LIN {X 0,Y 173.523,Z 389.647,A -85,B 0,C 180,E1 -26312.819,E2 -26312.819} C_VEL
LIN {X 0,Y 168.462,Z 401.528,A -85,B 0,C 180,E1 -26313.99,E2 -26313.99} C_VEL
LIN {X 0,Y 162.813,Z 412.302,A -85,B 0,C 180,E1 -26315.439,E2 -26315.439} C_VEL
LIN {X 0,Y 156.587,Z 422.141,A -85,B 0,C 180,E1 -26317.19,E2 -26317.19} C_VEL
LIN {X 0,Y 148.692,Z 432.687,A -85,B 0,C 180,E1 -26319.822,E2 -26319.822} C_VEL
LIN {X 0,Y 142.367,Z 439.895,A -85,B 0,C 180,E1 -26322.229,E2 -26322.229} C_VEL
LIN {X 0,Y 135.332,Z 447.062,A -85,B 0,C 180,E1 -26325.488,E2 -26325.488} C_VEL
LIN {X 0,Y 128.764,Z 452.875,A -85,B 0,C 180,E1 -26329.084,E2 -26329.084} C_VEL
LIN {X 0,Y 122.651,Z 457.744,A -85,B 0,C 180,E1 -26333.368,E2 -26333.368} C_VEL
LIN {X 0,Y 117.792,Z 461.088,A -85,B 0,C 180,E1 -26337.523,E2 -26337.523} C_VEL
LIN {X 0,Y 114.712,Z 462.976,A -85,B 0,C 180,E1 -26340.652,E2 -26340.652} C_VEL
LIN {X 0,Y 109.77,Z 465.505,A -85,B 0,C 180,E1 -26347.41,E2 -26347.41} C_VEL
LIN {X 0,Y 106.669,Z 466.55,A -85,B 0,C 180,E1 -26354.72,E2 -26354.72} C_VEL
LIN {X 0,Y 105.797,Z 466.508,A -85,B 0,C 180,E1 -26358.505,E2 -26358.505} C_VEL
LIN {X 0,Y 105.23,Z 465.234,A -85,B 0,C 180,E1 -26366.171,E2 -26366.171} C_VEL
LIN {X 0,Y 105.415,Z 464.016,A -85,B 0,C 180,E1 -26370,E2 -26370} C_VEL
LIN {X 0,Y 105.329,Z 461.286,A -85,B 0,C 180,E1 -26375.744,E2 -26375.744} C_VEL
LIN {X 0,Y 105.868,Z 457.47,A -85,B 0,C 180,E1 -26381.487,E2 -26381.487} C_VEL
LIN {X 0,Y 107.202,Z 452.472,A -85,B 0,C 180,E1 -26387.158,E2 -26387.158} C_VEL
LIN {X 0,Y 109.577,Z 446.168,A -85,B 0,C 180,E1 -26392.633,E2 -26392.633} C_VEL
LIN {X 0,Y 112.757,Z 438.217,A -85,B 0,C 180,E1 -26397.869,E2 -26397.869} C_VEL
LIN {X 0,Y 116.232,Z 429.754,A -85,B 0,C 180,E1 -26402.134,E2 -26402.134} C_VEL
LIN {X 0,Y 119.944,Z 420.166,A -85,B 0,C 180,E1 -26405.869,E2 -26405.869} C_VEL
LIN {X 0,Y 123.287,Z 410.655,A -85,B 0,C 180,E1 -26408.739,E2 -26408.739} C_VEL
LIN {X 0,Y 124.479,Z 405.7,A -85,B 0,C 180,E1 -26410.12,E2 -26410.12} C_VEL
LIN {X 0,Y 124.615,Z 397.297,A -85,B 0,C 180,E1 -26412.55,E2 -26412.55} C_VEL
LIN {X 0,Y 124.479,Z 388.532,A -85,B 0,C 180,E1 -26414.726,E2 -26414.726} C_VEL
LIN {X 0,Y 125.191,Z 382.999,A -85,B 0,C 180,E1 -26415.654,E2 -26415.654} C_VEL
LIN {X 0,Y 127.795,Z 369.185,A -85,B 0,C 180,E1 -26417.114,E2 -26417.114} C_VEL
LIN {X 0,Y 129.366,Z 355.732,A -85,B 0,C 180,E1 -26417.976,E2 -26417.976} C_VEL
LIN {X 0,Y 131.888,Z 324.068,A -85,B 0,C 180,E1 -26419.598,E2 -26419.598} C_VEL
LIN {X 0,Y 131.511,Z 321.043,A -85,B 0,C 180,E1 -26419.968,E2 -26419.968} C_VEL
LIN {X 0,Y 127.38,Z 308.413,A -85,B 0,C 180,E1 -26422.521,E2 -26422.521} C_VEL
LIN {X 0,Y 122.584,Z 296.227,A -85,B 0,C 180,E1 -26425.622,E2 -26425.622} C_VEL
LIN {X 0,Y 120.326,Z 291.293,A -85,B 0,C 180,E1 -26427.153,E2 -26427.153} C_VEL
LIN {X 0,Y 114.001,Z 280.829,A -85,B 0,C 180,E1 -26431.533,E2 -26431.533} C_VEL
LIN {X 0,Y 110.504,Z 275.927,A -85,B 0,C 180,E1 -26434.263,E2 -26434.263} C_VEL
LIN {X 0,Y 107.791,Z 271.993,A -85,B 0,C 180,E1 -26436.589,E2 -26436.589} C_VEL
LIN {X 0,Y 105.479,Z 269.052,A -85,B 0,C 180,E1 -26438.705,E2 -26438.705} C_VEL
LIN {X 0,Y 104.734,Z 267.39,A -85,B 0,C 180,E1 -26439.53,E2 -26439.53} C_VEL
LIN {X 0,Y 102.164,Z 265.254,A -85,B 0,C 180,E1 -26442.074,E2 -26442.074} C_VEL
LIN {X 0,Y 101.014,Z 262.807,A -85,B 0,C 180,E1 -26443.559,E2 -26443.559} C_VEL
LIN {X 0,Y 100.884,Z 261.872,A -85,B 0,C 180,E1 -26444.046,E2 -26444.046} C_VEL
LIN {X 0,Y 101.128,Z 261.886,A -85,B 0,C 180,E1 -26447.944,E2 -26447.944} C_VEL
LIN {X 0,Y 101.22,Z 261.842,A -85,B 0,C 180,E1 -26451.996,E2 -26451.996} C_VEL
LIN {X 0,Y 101.789,Z 261.752,A -85,B 0,C 180,E1 -26459.978,E2 -26459.978} C_VEL
LIN {X 0,Y 101.212,Z 261.861,A -85,B 0,C 180,E1 -26467.96,E2 -26467.96} C_VEL
LIN {X 0,Y 101.061,Z 261.894,A -85,B 0,C 180,E1 -26473.202,E2 -26473.202} C_VEL
LIN {X 0,Y 100.79,Z 261.914,A -85,B 0,C 180,E1 -26480.379,E2 -26480.379} C_VEL
LIN {X 0,Y 100.755,Z 261.924,A -85,B 0,C 180,E1 -26484.937,E2 -26484.937} C_VEL
LIN {X 0,Y 100.661,Z 261.873,A -85,B 0,C 180,E1 -26493.091,E2 -26493.091} C_VEL
LIN {X 0,Y 100.601,Z 261.954,A -85,B 0,C 180,E1 -26499.785,E2 -26499.785} C_VEL
LIN {X 0,Y 100.603,Z 261.947,A -85,B 0,C 180,E1 -26505.688,E2 -26505.688} C_VEL
LIN {X 0,Y 100.593,Z 261.97,A -85,B 0,C 180,E1 -26509.57,E2 -26509.57} C_VEL
LIN {X 0,Y 101.292,Z 264.266,A -85,B 0,C 180,E1 -26510.615,E2 -26510.615} C_VEL
LIN {X 0,Y 103.285,Z 266.68,A -85,B 0,C 180,E1 -26512.808,E2 -26512.808} C_VEL
LIN {X 0,Y 104.738,Z 267.806,A -85,B 0,C 180,E1 -26514.201,E2 -26514.201} C_VEL
LIN {X 0,Y 106.727,Z 271.057,A -85,B 0,C 180,E1 -26516.195,E2 -26516.195} C_VEL
LIN {X 0,Y 108.388,Z 272.818,A -85,B 0,C 180,E1 -26517.618,E2 -26517.618} C_VEL
LIN {X 0,Y 111.076,Z 276.52,A -85,B 0,C 180,E1 -26519.848,E2 -26519.848} C_VEL
LIN {X 0,Y 116.537,Z 284.607,A -85,B 0,C 180,E1 -26523.96,E2 -26523.96} C_VEL
LIN {X 0,Y 124.075,Z 297.45,A -85,B 0,C 180,E1 -26528.822,E2 -26528.822} C_VEL
LIN {X 0,Y 128.647,Z 306.796,A -85,B 0,C 180,E1 -26531.51,E2 -26531.51} C_VEL
LIN {X 0,Y 132.471,Z 314.86,A -85,B 0,C 180,E1 -26533.561,E2 -26533.561} C_VEL
LIN {X 0,Y 128.797,Z 356.517,A -85,B 0,C 180,E1 -26535.699,E2 -26535.699} C_VEL
LIN {X 0,Y 126.812,Z 369.27,A -85,B 0,C 180,E1 -26536.834,E2 -26536.834} C_VEL
LIN {X 0,Y 124.228,Z 382.01,A -85,B 0,C 180,E1 -26538.58,E2 -26538.58} C_VEL
LIN {X 0,Y 120.987,Z 393.79,A -85,B 0,C 180,E1 -26540.794,E2 -26540.794} C_VEL
LIN {X 0,Y 117.394,Z 404.765,A -85,B 0,C 180,E1 -26543.555,E2 -26543.555} C_VEL
LIN {X 0,Y 113.496,Z 415.135,A -85,B 0,C 180,E1 -26546.974,E2 -26546.974} C_VEL
LIN {X 0,Y 109.635,Z 424.292,A -85,B 0,C 180,E1 -26550.918,E2 -26550.918} C_VEL
LIN {X 0,Y 105.914,Z 432.882,A -85,B 0,C 180,E1 -26555.789,E2 -26555.789} C_VEL
LIN {X 0,Y 102.45,Z 440.996,A -85,B 0,C 180,E1 -26561.876,E2 -26561.876} C_VEL
LIN {X 0,Y 99.946,Z 447.442,A -85,B 0,C 180,E1 -26568.446,E2 -26568.446} C_VEL
LIN {X 0,Y 98.956,Z 450.682,A -85,B 0,C 180,E1 -26572.657,E2 -26572.657} C_VEL
LIN {X 0,Y 97.726,Z 455.179,A -85,B 0,C 180,E1 -26580.399,E2 -26580.399} C_VEL
LIN {X 0,Y 97.898,Z 457.999,A -85,B 0,C 180,E1 -26587.887,E2 -26587.887} C_VEL
LIN {X 0,Y 99.421,Z 459.479,A -85,B 0,C 180,E1 -26595.053,E2 -26595.053} C_VEL
LIN {X 0,Y 102.075,Z 459.766,A -85,B 0,C 180,E1 -26601.74,E2 -26601.74} C_VEL
LIN {X 0,Y 106.604,Z 458.714,A -85,B 0,C 180,E1 -26608.982,E2 -26608.982} C_VEL
LIN {X 0,Y 110.55,Z 457.11,A -85,B 0,C 180,E1 -26613.601,E2 -26613.601} C_VEL
LIN {X 0,Y 116.24,Z 454.155,A -85,B 0,C 180,E1 -26618.752,E2 -26618.752} C_VEL
LIN {X 0,Y 124.153,Z 449.027,A -85,B 0,C 180,E1 -26624.217,E2 -26624.217} C_VEL
LIN {X 0,Y 131.103,Z 443.664,A -85,B 0,C 180,E1 -26628.032,E2 -26628.032} C_VEL
LIN {X 0,Y 139.371,Z 436.152,A -85,B 0,C 180,E1 -26631.793,E2 -26631.793} C_VEL
LIN {X 0,Y 146.945,Z 427.927,A -85,B 0,C 180,E1 -26634.697,E2 -26634.697} C_VEL
LIN {X 0,Y 154.789,Z 417.865,A -85,B 0,C 180,E1 -26637.251,E2 -26637.251} C_VEL
LIN {X 0,Y 161.652,Z 407.117,A -85,B 0,C 180,E1 -26639.275,E2 -26639.275} C_VEL
LIN {X 0,Y 168.063,Z 394.85,A -85,B 0,C 180,E1 -26640.932,E2 -26640.932} C_VEL
LIN {X 0,Y 172.838,Z 383.164,A -85,B 0,C 180,E1 -26642.093,E2 -26642.093} C_VEL
LIN {X 0,Y 176.914,Z 369.735,A -85,B 0,C 180,E1 -26643.068,E2 -26643.068} C_VEL
LIN {X 0,Y 179.697,Z 356.281,A -85,B 0,C 180,E1 -26643.666,E2 -26643.666} C_VEL
LIN {X 0,Y 180.613,Z 349.351,A -85,B 0,C 180,E1 -26643.913,E2 -26643.913} C_VEL
LIN {X 0,Y 178.757,Z 344.448,A -85,B 0,C 180,E1 -26647.527,E2 -26647.527} C_VEL
LIN {X 0,Y 177.257,Z 340.928,A -85,B 0,C 180,E1 -26652.331,E2 -26652.331} C_VEL
LIN {X 0,Y 176.949,Z 340.868,A -85,B 0,C 180,E1 -26658.539,E2 -26658.539} C_VEL
LIN {X 0,Y 177.227,Z 341.36,A -85,B 0,C 180,E1 -26660.296,E2 -26660.296} C_VEL
LIN {X 0,Y 178.252,Z 345.016,A -85,B 0,C 180,E1 -26664.172,E2 -26664.172} C_VEL
LIN {X 0,Y 179.398,Z 349.511,A -85,B 0,C 180,E1 -26667.056,E2 -26667.056} C_VEL
LIN {X 0,Y 180.251,Z 352.766,A -85,B 0,C 180,E1 -26668.724,E2 -26668.724} C_VEL
LIN {X 0,Y 178.035,Z 366.835,A -85,B 0,C 180,E1 -26669.263,E2 -26669.263} C_VEL
LIN {X 0,Y 174.869,Z 379.037,A -85,B 0,C 180,E1 -26669.87,E2 -26669.87} C_VEL
LIN {X 0,Y 170.606,Z 391.041,A -85,B 0,C 180,E1 -26670.694,E2 -26670.694} C_VEL
LIN {X 0,Y 165.407,Z 402.543,A -85,B 0,C 180,E1 -26671.815,E2 -26671.815} C_VEL
LIN {X 0,Y 158.87,Z 414.143,A -85,B 0,C 180,E1 -26673.389,E2 -26673.389} C_VEL
LIN {X 0,Y 152.479,Z 423.6,A -85,B 0,C 180,E1 -26675.105,E2 -26675.105} C_VEL
LIN {X 0,Y 145.649,Z 432.274,A -85,B 0,C 180,E1 -26677.236,E2 -26677.236} C_VEL
LIN {X 0,Y 137.736,Z 440.839,A -85,B 0,C 180,E1 -26680.062,E2 -26680.062} C_VEL
LIN {X 0,Y 130.397,Z 447.728,A -85,B 0,C 180,E1 -26683.316,E2 -26683.316} C_VEL
LIN {X 0,Y 123.494,Z 453.321,A -85,B 0,C 180,E1 -26686.93,E2 -26686.93} C_VEL
LIN {X 0,Y 116.701,Z 458.231,A -85,B 0,C 180,E1 -26691.553,E2 -26691.553} C_VEL
LIN {X 0,Y 111.875,Z 461.26,A -85,B 0,C 180,E1 -26695.573,E2 -26695.573} C_VEL
LIN {X 0,Y 108.563,Z 463.024,A -85,B 0,C 180,E1 -26698.81,E2 -26698.81} C_VEL
LIN {X 0,Y 103.244,Z 465.403,A -85,B 0,C 180,E1 -26705.895,E2 -26705.895} C_VEL
LIN {X 0,Y 99.802,Z 466.291,A -85,B 0,C 180,E1 -26713.64,E2 -26713.64} C_VEL
LIN {X 0,Y 98.268,Z 465.638,A -85,B 0,C 180,E1 -26721.777,E2 -26721.777} C_VEL
LIN {X 0,Y 98.14,Z 464.75,A -85,B 0,C 180,E1 -26725.894,E2 -26725.894} C_VEL
LIN {X 0,Y 98.339,Z 463.468,A -85,B 0,C 180,E1 -26730,E2 -26730} C_VEL
LIN {X 0,Y 98.261,Z 460.606,A -85,B 0,C 180,E1 -26736.159,E2 -26736.159} C_VEL
LIN {X 0,Y 98.904,Z 456.656,A -85,B 0,C 180,E1 -26742.308,E2 -26742.308} C_VEL
LIN {X 0,Y 100.747,Z 450.496,A -85,B 0,C 180,E1 -26749.351,E2 -26749.351} C_VEL
LIN {X 0,Y 103.525,Z 443.746,A -85,B 0,C 180,E1 -26755.105,E2 -26755.105} C_VEL
LIN {X 0,Y 107.123,Z 435.315,A -85,B 0,C 180,E1 -26760.56,E2 -26760.56} C_VEL
LIN {X 0,Y 110.873,Z 426.629,A -85,B 0,C 180,E1 -26764.784,E2 -26764.784} C_VEL
LIN {X 0,Y 115.059,Z 415.888,A -85,B 0,C 180,E1 -26768.761,E2 -26768.761} C_VEL
LIN {X 0,Y 118.941,Z 405.316,A -85,B 0,C 180,E1 -26771.661,E2 -26771.661} C_VEL
LIN {X 0,Y 122.526,Z 393.559,A -85,B 0,C 180,E1 -26774.064,E2 -26774.064} C_VEL
LIN {X 0,Y 125.191,Z 382.999,A -85,B 0,C 180,E1 -26775.654,E2 -26775.654} C_VEL
LIN {X 0,Y 125.895,Z 377.401,A -85,B 0,C 180,E1 -26776.473,E2 -26776.473} C_VEL
LIN {X 0,Y 125.185,Z 368.17,A -85,B 0,C 180,E1 -26778.111,E2 -26778.111} C_VEL
LIN {X 0,Y 123.997,Z 358.801,A -85,B 0,C 180,E1 -26779.566,E2 -26779.566} C_VEL
LIN {X 0,Y 123.958,Z 352.975,A -85,B 0,C 180,E1 -26780.083,E2 -26780.083} C_VEL
LIN {X 0,Y 126.361,Z 325.409,A -85,B 0,C 180,E1 -26781.488,E2 -26781.488} C_VEL
LIN {X 0,Y 125.921,Z 322.704,A -85,B 0,C 180,E1 -26781.886,E2 -26781.886} C_VEL
LIN {X 0,Y 121.985,Z 310.518,A -85,B 0,C 180,E1 -26784.581,E2 -26784.581} C_VEL
LIN {X 0,Y 116.954,Z 297.511,A -85,B 0,C 180,E1 -26788.196,E2 -26788.196} C_VEL
LIN {X 0,Y 111.914,Z 288.646,A -85,B 0,C 180,E1 -26791.904,E2 -26791.904} C_VEL
LIN {X 0,Y 107.287,Z 281.615,A -85,B 0,C 180,E1 -26795.744,E2 -26795.744} C_VEL
LIN {X 0,Y 104.365,Z 277.426,A -85,B 0,C 180,E1 -26798.448,E2 -26798.448} C_VEL
LIN {X 0,Y 102.046,Z 273.886,A -85,B 0,C 180,E1 -26800.883,E2 -26800.883} C_VEL
LIN {X 0,Y 99.038,Z 270.451,A -85,B 0,C 180,E1 -26804.28,E2 -26804.28} C_VEL
LIN {X 0,Y 98.004,Z 268.327,A -85,B 0,C 180,E1 -26805.706,E2 -26805.706} C_VEL
LIN {X 0,Y 95.358,Z 266.042,A -85,B 0,C 180,E1 -26809.224,E2 -26809.224} C_VEL
LIN {X 0,Y 94.308,Z 263.664,A -85,B 0,C 180,E1 -26811.135,E2 -26811.135} C_VEL
LIN {X 0,Y 94.159,Z 262.723,A -85,B 0,C 180,E1 -26811.661,E2 -26811.661} C_VEL
LIN {X 0,Y 94.722,Z 262.629,A -85,B 0,C 180,E1 -26819.976,E2 -26819.976} C_VEL
LIN {X 0,Y 94.123,Z 262.74,A -85,B 0,C 180,E1 -26828.563,E2 -26828.563} C_VEL
LIN {X 0,Y 93.99,Z 262.776,A -85,B 0,C 180,E1 -26833.581,E2 -26833.581} C_VEL
LIN {X 0,Y 93.671,Z 262.812,A -85,B 0,C 180,E1 -26842.006,E2 -26842.006} C_VEL
LIN {X 0,Y 93.597,Z 262.785,A -85,B 0,C 180,E1 -26846.748,E2 -26846.748} C_VEL
LIN {X 0,Y 93.556,Z 262.764,A -85,B 0,C 180,E1 -26854.278,E2 -26854.278} C_VEL
LIN {X 0,Y 93.495,Z 262.855,A -85,B 0,C 180,E1 -26861.125,E2 -26861.125} C_VEL
LIN {X 0,Y 94.283,Z 265.311,A -85,B 0,C 180,E1 -26862.822,E2 -26862.822} C_VEL
LIN {X 0,Y 96.779,Z 267.956,A -85,B 0,C 180,E1 -26866.53,E2 -26866.53} C_VEL
LIN {X 0,Y 97.995,Z 268.816,A -85,B 0,C 180,E1 -26868.041,E2 -26868.041} C_VEL
LIN {X 0,Y 99.878,Z 272.01,A -85,B 0,C 180,E1 -26870.478,E2 -26870.478} C_VEL
LIN {X 0,Y 102.045,Z 274.168,A -85,B 0,C 180,E1 -26872.823,E2 -26872.823} C_VEL
LIN {X 0,Y 104.47,Z 277.68,A -85,B 0,C 180,E1 -26875.347,E2 -26875.347} C_VEL
LIN {X 0,Y 105.749,Z 279.442,A -85,B 0,C 180,E1 -26876.56,E2 -26876.56} C_VEL
LIN {X 0,Y 108.647,Z 283.578,A -85,B 0,C 180,E1 -26879.106,E2 -26879.106} C_VEL
LIN {X 0,Y 112.777,Z 289.788,A -85,B 0,C 180,E1 -26882.403,E2 -26882.403} C_VEL
LIN {X 0,Y 119.764,Z 302.011,A -85,B 0,C 180,E1 -26887.283,E2 -26887.283} C_VEL
LIN {X 0,Y 124.133,Z 311.337,A -85,B 0,C 180,E1 -26890.082,E2 -26890.082} C_VEL
LIN {X 0,Y 126.852,Z 317.258,A -85,B 0,C 180,E1 -26891.69,E2 -26891.69} C_VEL
LIN {X 0,Y 123.132,Z 356.805,A -85,B 0,C 180,E1 -26893.738,E2 -26893.738} C_VEL
LIN {X 0,Y 121.132,Z 369.242,A -85,B 0,C 180,E1 -26894.866,E2 -26894.866} C_VEL
LIN {X 0,Y 118.645,Z 381.15,A -85,B 0,C 180,E1 -26896.512,E2 -26896.512} C_VEL
LIN {X 0,Y 115.127,Z 393.617,A -85,B 0,C 180,E1 -26898.866,E2 -26898.866} C_VEL
LIN {X 0,Y 111.182,Z 405.069,A -85,B 0,C 180,E1 -26901.822,E2 -26901.822} C_VEL
LIN {X 0,Y 107.195,Z 415.209,A -85,B 0,C 180,E1 -26905.299,E2 -26905.299} C_VEL
LIN {X 0,Y 103.407,Z 423.789,A -85,B 0,C 180,E1 -26909.105,E2 -26909.105} C_VEL
LIN {X 0,Y 99.512,Z 432.289,A -85,B 0,C 180,E1 -26914.05,E2 -26914.05} C_VEL
LIN {X 0,Y 95.731,Z 440.649,A -85,B 0,C 180,E1 -26920.575,E2 -26920.575} C_VEL
LIN {X 0,Y 93.634,Z 445.644,A -85,B 0,C 180,E1 -26925.685,E2 -26925.685} C_VEL
LIN {X 0,Y 91.827,Z 450.816,A -85,B 0,C 180,E1 -26932.499,E2 -26932.499} C_VEL
LIN {X 0,Y 90.895,Z 453.817,A -85,B 0,C 180,E1 -26937.639,E2 -26937.639} C_VEL
LIN {X 0,Y 90.535,Z 456.209,A -85,B 0,C 180,E1 -26942.913,E2 -26942.913} C_VEL
LIN {X 0,Y 91.013,Z 458.358,A -85,B 0,C 180,E1 -26949.492,E2 -26949.492} C_VEL
LIN {X 0,Y 92.867,Z 459.787,A -85,B 0,C 180,E1 -26957.107,E2 -26957.107} C_VEL
LIN {X 0,Y 95.936,Z 460.045,A -85,B 0,C 180,E1 -26964.154,E2 -26964.154} C_VEL
LIN {X 0,Y 100.192,Z 459.213,A -85,B 0,C 180,E1 -26970.621,E2 -26970.621} C_VEL
LIN {X 0,Y 106.521,Z 456.851,A -85,B 0,C 180,E1 -26977.467,E2 -26977.467} C_VEL
LIN {X 0,Y 113.832,Z 453.141,A -85,B 0,C 180,E1 -26983.2,E2 -26983.2} C_VEL
LIN {X 0,Y 122.061,Z 447.923,A -85,B 0,C 180,E1 -26988.179,E2 -26988.179} C_VEL
LIN {X 0,Y 129.579,Z 442.176,A -85,B 0,C 180,E1 -26991.808,E2 -26991.808} C_VEL
LIN {X 0,Y 137.573,Z 434.944,A -85,B 0,C 180,E1 -26995.058,E2 -26995.058} C_VEL
LIN {X 0,Y 145.153,Z 426.943,A -85,B 0,C 180,E1 -26997.644,E2 -26997.644} C_VEL
LIN {X 0,Y 152.348,Z 417.995,A -85,B 0,C 180,E1 -26999.776,E2 -26999.776} C_VEL
LIN {X 0,Y 159.067,Z 407.882,A -85,B 0,C 180,E1 -27001.619,E2 -27001.619} C_VEL
LIN {X 0,Y 165.421,Z 396.229,A -85,B 0,C 180,E1 -27003.142,E2 -27003.142} C_VEL
LIN {X 0,Y 170.673,Z 384.025,A -85,B 0,C 180,E1 -27004.321,E2 -27004.321} C_VEL
LIN {X 0,Y 174.831,Z 370.891,A -85,B 0,C 180,E1 -27005.249,E2 -27005.249} C_VEL
LIN {X 0,Y 177.74,Z 357.732,A -85,B 0,C 180,E1 -27005.826,E2 -27005.826} C_VEL
LIN {X 0,Y 178.27,Z 353.981,A -85,B 0,C 180,E1 -27005.99,E2 -27005.99} C_VEL
LIN {X 0,Y 177.321,Z 350.885,A -85,B 0,C 180,E1 -27008.453,E2 -27008.453} C_VEL
LIN {X 0,Y 176.224,Z 348.004,A -85,B 0,C 180,E1 -27012.405,E2 -27012.405} C_VEL
LIN {X 0,Y 175.764,Z 347.739,A -85,B 0,C 180,E1 -27016.338,E2 -27016.338} C_VEL
LIN {X 0,Y 176.135,Z 348.278,A -85,B 0,C 180,E1 -27019.872,E2 -27019.872} C_VEL
LIN {X 0,Y 176.89,Z 351.495,A -85,B 0,C 180,E1 -27023.318,E2 -27023.318} C_VEL
LIN {X 0,Y 177.748,Z 355.653,A -85,B 0,C 180,E1 -27026.029,E2 -27026.029} C_VEL
LIN {X 0,Y 177.989,Z 356.648,A -85,B 0,C 180,E1 -27026.615,E2 -27026.615} C_VEL
LIN {X 0,Y 175.417,Z 370.297,A -85,B 0,C 180,E1 -27027.187,E2 -27027.187} C_VEL
LIN {X 0,Y 171.638,Z 383.047,A -85,B 0,C 180,E1 -27027.85,E2 -27027.85} C_VEL
LIN {X 0,Y 166.407,Z 395.955,A -85,B 0,C 180,E1 -27028.798,E2 -27028.798} C_VEL
LIN {X 0,Y 160.349,Z 407.721,A -85,B 0,C 180,E1 -27030.048,E2 -27030.048} C_VEL
LIN {X 0,Y 152.944,Z 419.266,A -85,B 0,C 180,E1 -27031.78,E2 -27031.78} C_VEL
LIN {X 0,Y 145.739,Z 428.632,A -85,B 0,C 180,E1 -27033.713,E2 -27033.713} C_VEL
LIN {X 0,Y 137.337,Z 437.79,A -85,B 0,C 180,E1 -27036.297,E2 -27036.297} C_VEL
LIN {X 0,Y 132.034,Z 442.9,A -85,B 0,C 180,E1 -27038.27,E2 -27038.27} C_VEL
LIN {X 0,Y 123.203,Z 450.326,A -85,B 0,C 180,E1 -27042.136,E2 -27042.136} C_VEL
LIN {X 0,Y 116.174,Z 455.352,A -85,B 0,C 180,E1 -27045.919,E2 -27045.919} C_VEL
LIN {X 0,Y 107.972,Z 460.382,A -85,B 0,C 180,E1 -27051.805,E2 -27051.805} C_VEL
LIN {X 0,Y 102.546,Z 463.065,A -85,B 0,C 180,E1 -27056.752,E2 -27056.752} C_VEL
LIN {X 0,Y 96.804,Z 465.306,A -85,B 0,C 180,E1 -27064.177,E2 -27064.177} C_VEL
LIN {X 0,Y 92.984,Z 465.991,A -85,B 0,C 180,E1 -27072.403,E2 -27072.403} C_VEL
LIN {X 0,Y 91.235,Z 465.214,A -85,B 0,C 180,E1 -27081.138,E2 -27081.138} C_VEL
LIN {X 0,Y 91.07,Z 464.265,A -85,B 0,C 180,E1 -27085.574,E2 -27085.574} C_VEL
LIN {X 0,Y 91.248,Z 462.869,A -85,B 0,C 180,E1 -27090,E2 -27090} C_VEL
LIN {X 0,Y 91.216,Z 459.887,A -85,B 0,C 180,E1 -27096.637,E2 -27096.637} C_VEL
LIN {X 0,Y 91.972,Z 455.79,A -85,B 0,C 180,E1 -27103.253,E2 -27103.253} C_VEL
LIN {X 0,Y 94.049,Z 449.439,A -85,B 0,C 180,E1 -27110.79,E2 -27110.79} C_VEL
LIN {X 0,Y 97.095,Z 442.51,A -85,B 0,C 180,E1 -27116.897,E2 -27116.897} C_VEL
LIN {X 0,Y 101.038,Z 433.781,A -85,B 0,C 180,E1 -27122.62,E2 -27122.62} C_VEL
LIN {X 0,Y 105.062,Z 424.825,A -85,B 0,C 180,E1 -27127.016,E2 -27127.016} C_VEL
LIN {X 0,Y 109.087,Z 414.961,A -85,B 0,C 180,E1 -27130.715,E2 -27130.715} C_VEL
LIN {X 0,Y 113.19,Z 404.217,A -85,B 0,C 180,E1 -27133.689,E2 -27133.689} C_VEL
LIN {X 0,Y 116.973,Z 392.213,A -85,B 0,C 180,E1 -27136.135,E2 -27136.135} C_VEL
LIN {X 0,Y 120.089,Z 379.847,A -85,B 0,C 180,E1 -27137.944,E2 -27137.944} C_VEL
LIN {X 0,Y 122.467,Z 366.77,A -85,B 0,C 180,E1 -27139.235,E2 -27139.235} C_VEL
LIN {X 0,Y 123.958,Z 352.975,A -85,B 0,C 180,E1 -27140.083,E2 -27140.083} C_VEL
LIN {X 0,Y 124.007,Z 345.206,A -85,B 0,C 180,E1 -27140.717,E2 -27140.717} C_VEL
LIN {X 0,Y 123.126,Z 337.634,A -85,B 0,C 180,E1 -27141.704,E2 -27141.704} C_VEL
LIN {X 0,Y 120.025,Z 322.955,A -85,B 0,C 180,E1 -27144.311,E2 -27144.311} C_VEL
LIN {X 0,Y 116.312,Z 311.382,A -85,B 0,C 180,E1 -27147.144,E2 -27147.144} C_VEL
LIN {X 0,Y 112.23,Z 300.945,A -85,B 0,C 180,E1 -27150.367,E2 -27150.367} C_VEL
LIN {X 0,Y 106.883,Z 291.476,A -85,B 0,C 180,E1 -27154.805,E2 -27154.805} C_VEL
LIN {X 0,Y 101.701,Z 283.584,A -85,B 0,C 180,E1 -27159.764,E2 -27159.764} C_VEL
LIN {X 0,Y 98.778,Z 279.283,A -85,B 0,C 180,E1 -27163.11,E2 -27163.11} C_VEL
LIN {X 0,Y 96.331,Z 276.17,A -85,B 0,C 180,E1 -27166.16,E2 -27166.16} C_VEL
LIN {X 0,Y 95.421,Z 274.582,A -85,B 0,C 180,E1 -27167.494,E2 -27167.494} C_VEL
LIN {X 0,Y 92.875,Z 271.714,A -85,B 0,C 180,E1 -27171.422,E2 -27171.422} C_VEL
LIN {X 0,Y 91.987,Z 269.446,A -85,B 0,C 180,E1 -27173.318,E2 -27173.318} C_VEL
LIN {X 0,Y 89.589,Z 267.855,A -85,B 0,C 180,E1 -27178.008,E2 -27178.008} C_VEL
LIN {X 0,Y 88.449,Z 266.328,A -85,B 0,C 180,E1 -27181.112,E2 -27181.112} C_VEL
LIN {X 0,Y 87.123,Z 263.903,A -85,B 0,C 180,E1 -27186.373,E2 -27186.373} C_VEL
LIN {X 0,Y 87.066,Z 263.628,A -85,B 0,C 180,E1 -27186.928,E2 -27186.928} C_VEL
LIN {X 0,Y 86.883,Z 263.662,A -85,B 0,C 180,E1 -27194.016,E2 -27194.016} C_VEL
LIN {X 0,Y 86.61,Z 263.673,A -85,B 0,C 180,E1 -27198.911,E2 -27198.911} C_VEL
LIN {X 0,Y 86.607,Z 263.813,A -85,B 0,C 180,E1 -27205.08,E2 -27205.08} C_VEL
LIN {X 0,Y 87.45,Z 266.502,A -85,B 0,C 180,E1 -27209.787,E2 -27209.787} C_VEL
LIN {X 0,Y 90.733,Z 269.352,A -85,B 0,C 180,E1 -27218.257,E2 -27218.257} C_VEL
LIN {X 0,Y 91.493,Z 269.892,A -85,B 0,C 180,E1 -27219.673,E2 -27219.673} C_VEL
LIN {X 0,Y 92.992,Z 272.744,A -85,B 0,C 180,E1 -27222.623,E2 -27222.623} C_VEL
LIN {X 0,Y 95.691,Z 275.372,A -85,B 0,C 180,E1 -27226.646,E2 -27226.646} C_VEL
LIN {X 0,Y 97.92,Z 278.767,A -85,B 0,C 180,E1 -27229.654,E2 -27229.654} C_VEL
LIN {X 0,Y 99.584,Z 280.638,A -85,B 0,C 180,E1 -27231.553,E2 -27231.553} C_VEL
LIN {X 0,Y 102.896,Z 285.469,A -85,B 0,C 180,E1 -27235.164,E2 -27235.164} C_VEL
LIN {X 0,Y 105.939,Z 290.098,A -85,B 0,C 180,E1 -27238.062,E2 -27238.062} C_VEL
LIN {X 0,Y 109.381,Z 295.454,A -85,B 0,C 180,E1 -27240.974,E2 -27240.974} C_VEL
LIN {X 0,Y 115.704,Z 307.061,A -85,B 0,C 180,E1 -27245.805,E2 -27245.805} C_VEL
LIN {X 0,Y 119.528,Z 315.472,A -85,B 0,C 180,E1 -27248.434,E2 -27248.434} C_VEL
LIN {X 0,Y 121.267,Z 319.451,A -85,B 0,C 180,E1 -27249.58,E2 -27249.58} C_VEL
LIN {X 0,Y 117.761,Z 356.34,A -85,B 0,C 180,E1 -27251.547,E2 -27251.547} C_VEL
LIN {X 0,Y 115.543,Z 369.586,A -85,B 0,C 180,E1 -27252.751,E2 -27252.751} C_VEL
LIN {X 0,Y 112.933,Z 381.47,A -85,B 0,C 180,E1 -27254.433,E2 -27254.433} C_VEL
LIN {X 0,Y 109.223,Z 393.936,A -85,B 0,C 180,E1 -27256.84,E2 -27256.84} C_VEL
LIN {X 0,Y 105.11,Z 405.361,A -85,B 0,C 180,E1 -27259.891,E2 -27259.891} C_VEL
LIN {X 0,Y 100.892,Z 415.494,A -85,B 0,C 180,E1 -27263.5,E2 -27263.5} C_VEL
LIN {X 0,Y 96.503,Z 424.847,A -85,B 0,C 180,E1 -27267.913,E2 -27267.913} C_VEL
LIN {X 0,Y 92.395,Z 433.306,A -85,B 0,C 180,E1 -27273.27,E2 -27273.27} C_VEL
LIN {X 0,Y 88.48,Z 441.531,A -85,B 0,C 180,E1 -27280.295,E2 -27280.295} C_VEL
LIN {X 0,Y 86.085,Z 447.029,A -85,B 0,C 180,E1 -27286.6,E2 -27286.6} C_VEL
LIN {X 0,Y 84.227,Z 452.27,A -85,B 0,C 180,E1 -27294.657,E2 -27294.657} C_VEL
LIN {X 0,Y 83.462,Z 456.015,A -85,B 0,C 180,E1 -27302.697,E2 -27302.697} C_VEL
LIN {X 0,Y 84.262,Z 458.834,A -85,B 0,C 180,E1 -27311.854,E2 -27311.854} C_VEL
LIN {X 0,Y 86.43,Z 460.095,A -85,B 0,C 180,E1 -27319.457,E2 -27319.457} C_VEL
LIN {X 0,Y 90.853,Z 460.228,A -85,B 0,C 180,E1 -27328.308,E2 -27328.308} C_VEL
LIN {X 0,Y 94.75,Z 459.48,A -85,B 0,C 180,E1 -27333.602,E2 -27333.602} C_VEL
LIN {X 0,Y 100.589,Z 457.58,A -85,B 0,C 180,E1 -27339.578,E2 -27339.578} C_VEL
LIN {X 0,Y 108.763,Z 453.849,A -85,B 0,C 180,E1 -27345.75,E2 -27345.75} C_VEL
LIN {X 0,Y 117.529,Z 448.737,A -85,B 0,C 180,E1 -27350.769,E2 -27350.769} C_VEL
LIN {X 0,Y 126.988,Z 441.945,A -85,B 0,C 180,E1 -27354.978,E2 -27354.978} C_VEL
LIN {X 0,Y 135.364,Z 434.691,A -85,B 0,C 180,E1 -27358.04,E2 -27358.04} C_VEL
LIN {X 0,Y 143.284,Z 426.551,A -85,B 0,C 180,E1 -27360.518,E2 -27360.518} C_VEL
LIN {X 0,Y 151.236,Z 416.725,A -85,B 0,C 180,E1 -27362.678,E2 -27362.678} C_VEL
LIN {X 0,Y 157.681,Z 407.129,A -85,B 0,C 180,E1 -27364.252,E2 -27364.252} C_VEL
LIN {X 0,Y 164.196,Z 395.395,A -85,B 0,C 180,E1 -27365.659,E2 -27365.659} C_VEL
LIN {X 0,Y 169.399,Z 383.338,A -85,B 0,C 180,E1 -27366.742,E2 -27366.742} C_VEL
LIN {X 0,Y 173.709,Z 369.902,A -85,B 0,C 180,E1 -27367.598,E2 -27367.598} C_VEL
LIN {X 0,Y 176.216,Z 358.691,A -85,B 0,C 180,E1 -27368.058,E2 -27368.058} C_VEL
LIN {X 0,Y 175.751,Z 357.293,A -85,B 0,C 180,E1 -27369.573,E2 -27369.573} C_VEL
LIN {X 0,Y 175.047,Z 354.907,A -85,B 0,C 180,E1 -27373.08,E2 -27373.08} C_VEL
LIN {X 0,Y 174.941,Z 354.954,A -85,B 0,C 180,E1 -27378.759,E2 -27378.759} C_VEL
LIN {X 0,Y 175.149,Z 356.181,A -85,B 0,C 180,E1 -27380.675,E2 -27380.675} C_VEL
LIN {X 0,Y 175.606,Z 358.717,A -85,B 0,C 180,E1 -27383.006,E2 -27383.006} C_VEL
LIN {X 0,Y 175.938,Z 360.875,A -85,B 0,C 180,E1 -27384.496,E2 -27384.496} C_VEL
LIN {X 0,Y 173.324,Z 372.495,A -85,B 0,C 180,E1 -27384.978,E2 -27384.978} C_VEL
LIN {X 0,Y 169.377,Z 384.723,A -85,B 0,C 180,E1 -27385.622,E2 -27385.622} C_VEL
LIN {X 0,Y 163.962,Z 397.316,A -85,B 0,C 180,E1 -27386.524,E2 -27386.524} C_VEL
LIN {X 0,Y 157.746,Z 408.654,A -85,B 0,C 180,E1 -27387.692,E2 -27387.692} C_VEL
LIN {X 0,Y 150.145,Z 419.999,A -85,B 0,C 180,E1 -27389.334,E2 -27389.334} C_VEL
LIN {X 0,Y 143.438,Z 428.338,A -85,B 0,C 180,E1 -27390.972,E2 -27390.972} C_VEL
LIN {X 0,Y 134.735,Z 437.492,A -85,B 0,C 180,E1 -27393.43,E2 -27393.43} C_VEL
LIN {X 0,Y 127.797,Z 443.777,A -85,B 0,C 180,E1 -27395.794,E2 -27395.794} C_VEL
LIN {X 0,Y 121.16,Z 449.032,A -85,B 0,C 180,E1 -27398.459,E2 -27398.459} C_VEL
LIN {X 0,Y 113.574,Z 454.255,A -85,B 0,C 180,E1 -27402.052,E2 -27402.052} C_VEL
LIN {X 0,Y 106.472,Z 458.503,A -85,B 0,C 180,E1 -27406.389,E2 -27406.389} C_VEL
LIN {X 0,Y 100.466,Z 461.52,A -85,B 0,C 180,E1 -27410.982,E2 -27410.982} C_VEL
LIN {X 0,Y 93.346,Z 464.343,A -85,B 0,C 180,E1 -27418.196,E2 -27418.196} C_VEL
LIN {X 0,Y 88.013,Z 465.603,A -85,B 0,C 180,E1 -27426.469,E2 -27426.469} C_VEL
LIN {X 0,Y 84.973,Z 465.42,A -85,B 0,C 180,E1 -27435.634,E2 -27435.634} C_VEL
LIN {X 0,Y 84.227,Z 464.771,A -85,B 0,C 180,E1 -27440.394,E2 -27440.394} C_VEL
LIN {X 0,Y 84.021,Z 463.708,A -85,B 0,C 180,E1 -27445.202,E2 -27445.202} C_VEL
LIN {X 0,Y 84.166,Z 462.238,A -85,B 0,C 180,E1 -27450,E2 -27450} C_VEL
LIN {X 0,Y 84.154,Z 459.119,A -85,B 0,C 180,E1 -27457.196,E2 -27457.196} C_VEL
LIN {X 0,Y 85.036,Z 454.878,A -85,B 0,C 180,E1 -27464.356,E2 -27464.356} C_VEL
LIN {X 0,Y 87.43,Z 448.381,A -85,B 0,C 180,E1 -27472.446,E2 -27472.446} C_VEL
LIN {X 0,Y 90.785,Z 441.216,A -85,B 0,C 180,E1 -27478.936,E2 -27478.936} C_VEL
LIN {X 0,Y 95.123,Z 432.242,A -85,B 0,C 180,E1 -27484.931,E2 -27484.931} C_VEL
LIN {X 0,Y 99.425,Z 423.019,A -85,B 0,C 180,E1 -27489.507,E2 -27489.507} C_VEL
LIN {X 0,Y 103.775,Z 412.763,A -85,B 0,C 180,E1 -27493.289,E2 -27493.289} C_VEL
LIN {X 0,Y 108.16,Z 401.508,A -85,B 0,C 180,E1 -27496.291,E2 -27496.291} C_VEL
LIN {X 0,Y 111.585,Z 390.866,A -85,B 0,C 180,E1 -27498.41,E2 -27498.41} C_VEL
LIN {X 0,Y 114.829,Z 378.085,A -85,B 0,C 180,E1 -27500.252,E2 -27500.252} C_VEL
LIN {X 0,Y 117.35,Z 363.993,A -85,B 0,C 180,E1 -27501.557,E2 -27501.557} C_VEL
LIN {X 0,Y 120.941,Z 326.088,A -85,B 0,C 180,E1 -27503.624,E2 -27503.624} C_VEL
LIN {X 0,Y 120.025,Z 322.955,A -85,B 0,C 180,E1 -27504.311,E2 -27504.311} C_VEL
LIN {X 0,Y 118.94,Z 319.584,A -85,B 0,C 180,E1 -27505.116,E2 -27505.116} C_VEL
LIN {X 0,Y 116.564,Z 315.198,A -85,B 0,C 180,E1 -27506.658,E2 -27506.658} C_VEL
LIN {X 0,Y 113.72,Z 311.448,A -85,B 0,C 180,E1 -27508.478,E2 -27508.478} C_VEL
LIN {X 0,Y 109.71,Z 306.766,A -85,B 0,C 180,E1 -27511.229,E2 -27511.229} C_VEL
LIN {X 0,Y 106.172,Z 301.687,A -85,B 0,C 180,E1 -27514.039,E2 -27514.039} C_VEL
LIN {X 0,Y 102.343,Z 295.138,A -85,B 0,C 180,E1 -27517.618,E2 -27517.618} C_VEL
LIN {X 0,Y 98.597,Z 289.101,A -85,B 0,C 180,E1 -27521.709,E2 -27521.709} C_VEL
LIN {X 0,Y 96.126,Z 285.335,A -85,B 0,C 180,E1 -27524.777,E2 -27524.777} C_VEL
LIN {X 0,Y 93.612,Z 281.66,A -85,B 0,C 180,E1 -27528.337,E2 -27528.337} C_VEL
LIN {X 0,Y 92.806,Z 280.57,A -85,B 0,C 180,E1 -27529.607,E2 -27529.607} C_VEL
LIN {X 0,Y 90.635,Z 277.549,A -85,B 0,C 180,E1 -27533.527,E2 -27533.527} C_VEL
LIN {X 0,Y 89.968,Z 276.094,A -85,B 0,C 180,E1 -27534.991,E2 -27534.991} C_VEL
LIN {X 0,Y 87.769,Z 274.123,A -85,B 0,C 180,E1 -27539.974,E2 -27539.974} C_VEL
LIN {X 0,Y 86.859,Z 272.85,A -85,B 0,C 180,E1 -27542.872,E2 -27542.872} C_VEL
LIN {X 0,Y 85.827,Z 270.642,A -85,B 0,C 180,E1 -27547.68,E2 -27547.68} C_VEL
LIN {X 0,Y 85.354,Z 270.688,A -85,B 0,C 180,E1 -27563.635,E2 -27563.635} C_VEL
LIN {X 0,Y 86.432,Z 273.718,A -85,B 0,C 180,E1 -27569.838,E2 -27569.838} C_VEL
LIN {X 0,Y 89.604,Z 276.525,A -85,B 0,C 180,E1 -27578.185,E2 -27578.185} C_VEL
LIN {X 0,Y 91.52,Z 279.774,A -85,B 0,C 180,E1 -27582.056,E2 -27582.056} C_VEL
LIN {X 0,Y 93.434,Z 281.753,A -85,B 0,C 180,E1 -27585.13,E2 -27585.13} C_VEL
LIN {X 0,Y 95.866,Z 285.322,A -85,B 0,C 180,E1 -27588.635,E2 -27588.635} C_VEL
LIN {X 0,Y 97.181,Z 287.14,A -85,B 0,C 180,E1 -27590.295,E2 -27590.295} C_VEL
LIN {X 0,Y 100.331,Z 291.885,A -85,B 0,C 180,E1 -27593.943,E2 -27593.943} C_VEL
LIN {X 0,Y 105.049,Z 299.359,A -85,B 0,C 180,E1 -27598.602,E2 -27598.602} C_VEL
LIN {X 0,Y 110.582,Z 309.828,A -85,B 0,C 180,E1 -27603.327,E2 -27603.327} C_VEL
LIN {X 0,Y 113.84,Z 316.737,A -85,B 0,C 180,E1 -27605.832,E2 -27605.832} C_VEL
LIN {X 0,Y 115.894,Z 321.712,A -85,B 0,C 180,E1 -27607.347,E2 -27607.347} C_VEL
LIN {X 0,Y 112.354,Z 356.852,A -85,B 0,C 180,E1 -27609.245,E2 -27609.245} C_VEL
LIN {X 0,Y 110.018,Z 370.26,A -85,B 0,C 180,E1 -27610.507,E2 -27610.507} C_VEL
LIN {X 0,Y 107.047,Z 382.759,A -85,B 0,C 180,E1 -27612.324,E2 -27612.324} C_VEL
LIN {X 0,Y 103.073,Z 395.247,A -85,B 0,C 180,E1 -27614.878,E2 -27614.878} C_VEL
LIN {X 0,Y 98.586,Z 406.906,A -85,B 0,C 180,E1 -27618.173,E2 -27618.173} C_VEL
LIN {X 0,Y 93.739,Z 417.543,A -85,B 0,C 180,E1 -27622.282,E2 -27622.282} C_VEL
LIN {X 0,Y 88.668,Z 427.75,A -85,B 0,C 180,E1 -27627.728,E2 -27627.728} C_VEL
LIN {X 0,Y 84.465,Z 435.885,A -85,B 0,C 180,E1 -27633.673,E2 -27633.673} C_VEL
LIN {X 0,Y 81.195,Z 442.349,A -85,B 0,C 180,E1 -27639.968,E2 -27639.968} C_VEL
LIN {X 0,Y 78.44,Z 448.674,A -85,B 0,C 180,E1 -27648.275,E2 -27648.275} C_VEL
LIN {X 0,Y 76.723,Z 453.647,A -85,B 0,C 180,E1 -27657.258,E2 -27657.258} C_VEL
LIN {X 0,Y 76.356,Z 456.407,A -85,B 0,C 180,E1 -27664.126,E2 -27664.126} C_VEL
LIN {X 0,Y 77.412,Z 459.038,A -85,B 0,C 180,E1 -27673.47,E2 -27673.47} C_VEL
LIN {X 0,Y 80.135,Z 460.393,A -85,B 0,C 180,E1 -27682.166,E2 -27682.166} C_VEL
LIN {X 0,Y 84.248,Z 460.606,A -85,B 0,C 180,E1 -27689.999,E2 -27689.999} C_VEL
LIN {X 0,Y 90.821,Z 459.433,A -85,B 0,C 180,E1 -27698.213,E2 -27698.213} C_VEL
LIN {X 0,Y 96.061,Z 457.829,A -85,B 0,C 180,E1 -27703.009,E2 -27703.009} C_VEL
LIN {X 0,Y 103.522,Z 454.782,A -85,B 0,C 180,E1 -27708.272,E2 -27708.272} C_VEL
LIN {X 0,Y 111.687,Z 450.528,A -85,B 0,C 180,E1 -27712.791,E2 -27712.791} C_VEL
LIN {X 0,Y 120.552,Z 444.868,A -85,B 0,C 180,E1 -27716.677,E2 -27716.677} C_VEL
LIN {X 0,Y 129.808,Z 437.705,A -85,B 0,C 180,E1 -27720.018,E2 -27720.018} C_VEL
LIN {X 0,Y 138.91,Z 429.19,A -85,B 0,C 180,E1 -27722.695,E2 -27722.695} C_VEL
LIN {X 0,Y 147.224,Z 419.815,A -85,B 0,C 180,E1 -27724.81,E2 -27724.81} C_VEL
LIN {X 0,Y 154.814,Z 409.455,A -85,B 0,C 180,E1 -27726.531,E2 -27726.531} C_VEL
LIN {X 0,Y 161.713,Z 397.746,A -85,B 0,C 180,E1 -27727.904,E2 -27727.904} C_VEL
LIN {X 0,Y 167.179,Z 386.042,A -85,B 0,C 180,E1 -27728.928,E2 -27728.928} C_VEL
LIN {X 0,Y 171.627,Z 373.394,A -85,B 0,C 180,E1 -27729.759,E2 -27729.759} C_VEL
LIN {X 0,Y 174.103,Z 363.98,A -85,B 0,C 180,E1 -27730.151,E2 -27730.151} C_VEL
LIN {X 0,Y 173.719,Z 361.876,A -85,B 0,C 180,E1 -27733.181,E2 -27733.181} C_VEL
LIN {X 0,Y 173.606,Z 361.902,A -85,B 0,C 180,E1 -27738.365,E2 -27738.365} C_VEL
LIN {X 0,Y 173.719,Z 362.623,A -85,B 0,C 180,E1 -27739.798,E2 -27739.798} C_VEL
LIN {X 0,Y 173.939,Z 365.359,A -85,B 0,C 180,E1 -27742.336,E2 -27742.336} C_VEL
LIN {X 0,Y 171.97,Z 373.114,A -85,B 0,C 180,E1 -27742.679,E2 -27742.679} C_VEL
LIN {X 0,Y 167.433,Z 386.468,A -85,B 0,C 180,E1 -27743.339,E2 -27743.339} C_VEL
LIN {X 0,Y 161.779,Z 398.737,A -85,B 0,C 180,E1 -27744.181,E2 -27744.181} C_VEL
LIN {X 0,Y 154.652,Z 410.977,A -85,B 0,C 180,E1 -27745.422,E2 -27745.422} C_VEL
LIN {X 0,Y 147.632,Z 420.778,A -85,B 0,C 180,E1 -27746.803,E2 -27746.803} C_VEL
LIN {X 0,Y 139.971,Z 429.716,A -85,B 0,C 180,E1 -27748.519,E2 -27748.519} C_VEL
LIN {X 0,Y 130.999,Z 438.538,A -85,B 0,C 180,E1 -27750.867,E2 -27750.867} C_VEL
LIN {X 0,Y 125.199,Z 443.503,A -85,B 0,C 180,E1 -27752.649,E2 -27752.649} C_VEL
LIN {X 0,Y 116.909,Z 449.706,A -85,B 0,C 180,E1 -27755.754,E2 -27755.754} C_VEL
LIN {X 0,Y 108.957,Z 454.725,A -85,B 0,C 180,E1 -27759.285,E2 -27759.285} C_VEL
LIN {X 0,Y 99.391,Z 459.749,A -85,B 0,C 180,E1 -27765.002,E2 -27765.002} C_VEL
LIN {X 0,Y 95.046,Z 461.664,A -85,B 0,C 180,E1 -27768.282,E2 -27768.282} C_VEL
LIN {X 0,Y 87.365,Z 464.264,A -85,B 0,C 180,E1 -27775.731,E2 -27775.731} C_VEL
LIN {X 0,Y 81.525,Z 465.373,A -85,B 0,C 180,E1 -27784.468,E2 -27784.468} C_VEL
LIN {X 0,Y 78.105,Z 465.032,A -85,B 0,C 180,E1 -27794.34,E2 -27794.34} C_VEL
LIN {X 0,Y 76.96,Z 463.136,A -85,B 0,C 180,E1 -27804.761,E2 -27804.761} C_VEL
LIN {X 0,Y 77.084,Z 461.597,A -85,B 0,C 180,E1 -27810,E2 -27810} C_VEL
LIN {X 0,Y 77.12,Z 458.328,A -85,B 0,C 180,E1 -27817.857,E2 -27817.857} C_VEL
LIN {X 0,Y 78.149,Z 453.925,A -85,B 0,C 180,E1 -27825.652,E2 -27825.652} C_VEL
LIN {X 0,Y 80.379,Z 448.274,A -85,B 0,C 180,E1 -27833.17,E2 -27833.17} C_VEL
LIN {X 0,Y 83.913,Z 441.173,A -85,B 0,C 180,E1 -27840.166,E2 -27840.166} C_VEL
LIN {X 0,Y 88.5,Z 432.258,A -85,B 0,C 180,E1 -27846.554,E2 -27846.554} C_VEL
LIN {X 0,Y 93.112,Z 422.977,A -85,B 0,C 180,E1 -27851.427,E2 -27851.427} C_VEL
LIN {X 0,Y 97.616,Z 412.968,A -85,B 0,C 180,E1 -27855.312,E2 -27855.312} C_VEL
LIN {X 0,Y 102.185,Z 401.829,A -85,B 0,C 180,E1 -27858.412,E2 -27858.412} C_VEL
LIN {X 0,Y 106.39,Z 389.41,A -85,B 0,C 180,E1 -27860.912,E2 -27860.912} C_VEL
LIN {X 0,Y 109.603,Z 376.756,A -85,B 0,C 180,E1 -27862.703,E2 -27862.703} C_VEL
LIN {X 0,Y 112.165,Z 362.936,A -85,B 0,C 180,E1 -27863.942,E2 -27863.942} C_VEL
LIN {X 0,Y 115.6,Z 327.888,A -85,B 0,C 180,E1 -27865.874,E2 -27865.874} C_VEL
LIN {X 0,Y 112.09,Z 316.117,A -85,B 0,C 180,E1 -27868.829,E2 -27868.829} C_VEL
LIN {X 0,Y 108.063,Z 305.254,A -85,B 0,C 180,E1 -27872.379,E2 -27872.379} C_VEL
LIN {X 0,Y 106.172,Z 301.687,A -85,B 0,C 180,E1 -27874.039,E2 -27874.039} C_VEL
LIN {X 0,Y 104.372,Z 299.54,A -85,B 0,C 180,E1 -27875.539,E2 -27875.539} C_VEL
LIN {X 0,Y 100.804,Z 297.694,A -85,B 0,C 180,E1 -27878.512,E2 -27878.512} C_VEL
LIN {X 0,Y 96.704,Z 295.768,A -85,B 0,C 180,E1 -27882.468,E2 -27882.468} C_VEL
LIN {X 0,Y 95.593,Z 294.584,A -85,B 0,C 180,E1 -27883.757,E2 -27883.757} C_VEL
LIN {X 0,Y 93.513,Z 291.283,A -85,B 0,C 180,E1 -27886.6,E2 -27886.6} C_VEL
LIN {X 0,Y 90.883,Z 287.098,A -85,B 0,C 180,E1 -27890.869,E2 -27890.869} C_VEL
LIN {X 0,Y 88.641,Z 283.837,A -85,B 0,C 180,E1 -27895.257,E2 -27895.257} C_VEL
LIN {X 0,Y 88.107,Z 282.732,A -85,B 0,C 180,E1 -27896.545,E2 -27896.545} C_VEL
LIN {X 0,Y 86.083,Z 280.383,A -85,B 0,C 180,E1 -27901.947,E2 -27901.947} C_VEL
LIN {X 0,Y 84.585,Z 277.596,A -85,B 0,C 180,E1 -27908.815,E2 -27908.815} C_VEL
LIN {X 0,Y 84.253,Z 277.786,A -85,B 0,C 180,E1 -27923.107,E2 -27923.107} C_VEL
LIN {X 0,Y 85.081,Z 280.458,A -85,B 0,C 180,E1 -27928.631,E2 -27928.631} C_VEL
LIN {X 0,Y 87.896,Z 283.323,A -85,B 0,C 180,E1 -27936.911,E2 -27936.911} C_VEL
LIN {X 0,Y 90.177,Z 286.885,A -85,B 0,C 180,E1 -27941.682,E2 -27941.682} C_VEL
LIN {X 0,Y 91.375,Z 288.355,A -85,B 0,C 180,E1 -27943.769,E2 -27943.769} C_VEL
LIN {X 0,Y 94.606,Z 293.216,A -85,B 0,C 180,E1 -27948.663,E2 -27948.663} C_VEL
LIN {X 0,Y 98.151,Z 298.739,A -85,B 0,C 180,E1 -27953.039,E2 -27953.039} C_VEL
LIN {X 0,Y 102.124,Z 305.612,A -85,B 0,C 180,E1 -27957.299,E2 -27957.299} C_VEL
LIN {X 0,Y 107.383,Z 316.053,A -85,B 0,C 180,E1 -27962.115,E2 -27962.115} C_VEL
LIN {X 0,Y 110.677,Z 324.066,A -85,B 0,C 180,E1 -27964.921,E2 -27964.921} C_VEL
LIN {X 0,Y 107.134,Z 357.373,A -85,B 0,C 180,E1 -27966.734,E2 -27966.734} C_VEL
LIN {X 0,Y 104.788,Z 370.317,A -85,B 0,C 180,E1 -27967.966,E2 -27967.966} C_VEL
LIN {X 0,Y 101.683,Z 382.791,A -85,B 0,C 180,E1 -27969.783,E2 -27969.783} C_VEL
LIN {X 0,Y 97.753,Z 394.666,A -85,B 0,C 180,E1 -27972.209,E2 -27972.209} C_VEL
LIN {X 0,Y 93.102,Z 406.258,A -85,B 0,C 180,E1 -27975.495,E2 -27975.495} C_VEL
LIN {X 0,Y 88.017,Z 416.975,A -85,B 0,C 180,E1 -27979.65,E2 -27979.65} C_VEL
LIN {X 0,Y 82.724,Z 427.021,A -85,B 0,C 180,E1 -27985.126,E2 -27985.126} C_VEL
LIN {X 0,Y 78.179,Z 435.273,A -85,B 0,C 180,E1 -27991.325,E2 -27991.325} C_VEL
LIN {X 0,Y 74.574,Z 441.965,A -85,B 0,C 180,E1 -27998.126,E2 -27998.126} C_VEL
LIN {X 0,Y 71.506,Z 448.43,A -85,B 0,C 180,E1 -28007.148,E2 -28007.148} C_VEL
LIN {X 0,Y 69.866,Z 452.716,A -85,B 0,C 180,E1 -28015.215,E2 -28015.215} C_VEL
LIN {X 0,Y 69.317,Z 456.773,A -85,B 0,C 180,E1 -28025.856,E2 -28025.856} C_VEL
LIN {X 0,Y 70.811,Z 459.365,A -85,B 0,C 180,E1 -28036.04,E2 -28036.04} C_VEL
LIN {X 0,Y 74.065,Z 460.692,A -85,B 0,C 180,E1 -28045.336,E2 -28045.336} C_VEL
LIN {X 0,Y 78.828,Z 460.887,A -85,B 0,C 180,E1 -28053.561,E2 -28053.561} C_VEL
LIN {X 0,Y 84.855,Z 460.018,A -85,B 0,C 180,E1 -28060.682,E2 -28060.682} C_VEL
LIN {X 0,Y 93.46,Z 457.568,A -85,B 0,C 180,E1 -28067.833,E2 -28067.833} C_VEL
LIN {X 0,Y 102.652,Z 453.828,A -85,B 0,C 180,E1 -28073.377,E2 -28073.377} C_VEL
LIN {X 0,Y 112.52,Z 448.603,A -85,B 0,C 180,E1 -28077.9,E2 -28077.9} C_VEL
LIN {X 0,Y 123.038,Z 441.598,A -85,B 0,C 180,E1 -28081.664,E2 -28081.664} C_VEL
LIN {X 0,Y 132.306,Z 434.062,A -85,B 0,C 180,E1 -28084.397,E2 -28084.397} C_VEL
LIN {X 0,Y 141.509,Z 424.928,A -85,B 0,C 180,E1 -28086.654,E2 -28086.654} C_VEL
LIN {X 0,Y 150.109,Z 414.546,A -85,B 0,C 180,E1 -28088.494,E2 -28088.494} C_VEL
LIN {X 0,Y 157.573,Z 403.351,A -85,B 0,C 180,E1 -28089.887,E2 -28089.887} C_VEL
LIN {X 0,Y 163.837,Z 391.653,A -85,B 0,C 180,E1 -28090.97,E2 -28090.97} C_VEL
LIN {X 0,Y 168.787,Z 379.783,A -85,B 0,C 180,E1 -28091.778,E2 -28091.778} C_VEL
LIN {X 0,Y 172.004,Z 369.573,A -85,B 0,C 180,E1 -28092.318,E2 -28092.318} C_VEL
LIN {X 0,Y 172.011,Z 368.741,A -85,B 0,C 180,E1 -28093.445,E2 -28093.445} C_VEL
LIN {X 0,Y 171.981,Z 368.843,A -85,B 0,C 180,E1 -28098.545,E2 -28098.545} C_VEL
LIN {X 0,Y 171.925,Z 370.401,A -85,B 0,C 180,E1 -28100.248,E2 -28100.248} C_VEL
LIN {X 0,Y 168.158,Z 382.084,A -85,B 0,C 180,E1 -28100.713,E2 -28100.713} C_VEL
LIN {X 0,Y 163.155,Z 393.759,A -85,B 0,C 180,E1 -28101.333,E2 -28101.333} C_VEL
LIN {X 0,Y 156.634,Z 405.784,A -85,B 0,C 180,E1 -28102.272,E2 -28102.272} C_VEL
LIN {X 0,Y 149.387,Z 416.507,A -85,B 0,C 180,E1 -28103.457,E2 -28103.457} C_VEL
LIN {X 0,Y 141.449,Z 426.167,A -85,B 0,C 180,E1 -28104.942,E2 -28104.942} C_VEL
LIN {X 0,Y 132.138,Z 435.607,A -85,B 0,C 180,E1 -28107.02,E2 -28107.02} C_VEL
LIN {X 0,Y 122.978,Z 443.265,A -85,B 0,C 180,E1 -28109.368,E2 -28109.368} C_VEL
LIN {X 0,Y 115.807,Z 448.47,A -85,B 0,C 180,E1 -28111.832,E2 -28111.832} C_VEL
LIN {X 0,Y 107.334,Z 453.685,A -85,B 0,C 180,E1 -28115.07,E2 -28115.07} C_VEL
LIN {X 0,Y 99.422,Z 457.792,A -85,B 0,C 180,E1 -28118.963,E2 -28118.963} C_VEL
LIN {X 0,Y 93.606,Z 460.353,A -85,B 0,C 180,E1 -28122.541,E2 -28122.541} C_VEL
LIN {X 0,Y 85.521,Z 463.164,A -85,B 0,C 180,E1 -28128.897,E2 -28128.897} C_VEL
LIN {X 0,Y 78.119,Z 464.846,A -85,B 0,C 180,E1 -28137.332,E2 -28137.332} C_VEL
LIN {X 0,Y 75.155,Z 465.14,A -85,B 0,C 180,E1 -28142.125,E2 -28142.125} C_VEL
LIN {X 0,Y 71.292,Z 464.584,A -85,B 0,C 180,E1 -28152.799,E2 -28152.799} C_VEL
LIN {X 0,Y 69.891,Z 462.555,A -85,B 0,C 180,E1 -28164.229,E2 -28164.229} C_VEL
LIN {X 0,Y 69.996,Z 460.943,A -85,B 0,C 180,E1 -28170,E2 -28170} C_VEL
LIN {X 0,Y 70.092,Z 457.533,A -85,B 0,C 180,E1 -28178.65,E2 -28178.65} C_VEL
LIN {X 0,Y 71.32,Z 452.964,A -85,B 0,C 180,E1 -28187.195,E2 -28187.195} C_VEL
LIN {X 0,Y 74.49,Z 445.98,A -85,B 0,C 180,E1 -28196.625,E2 -28196.625} C_VEL
LIN {X 0,Y 78.606,Z 438.387,A -85,B 0,C 180,E1 -28203.972,E2 -28203.972} C_VEL
LIN {X 0,Y 82.893,Z 430.61,A -85,B 0,C 180,E1 -28209.485,E2 -28209.485} C_VEL
LIN {X 0,Y 87.706,Z 421.298,A -85,B 0,C 180,E1 -28214.358,E2 -28214.358} C_VEL
LIN {X 0,Y 92.75,Z 410.527,A -85,B 0,C 180,E1 -28218.439,E2 -28218.439} C_VEL
LIN {X 0,Y 97.588,Z 398.884,A -85,B 0,C 180,E1 -28221.552,E2 -28221.552} C_VEL
LIN {X 0,Y 101.74,Z 386.579,A -85,B 0,C 180,E1 -28223.836,E2 -28223.836} C_VEL
LIN {X 0,Y 105.004,Z 373.521,A -85,B 0,C 180,E1 -28225.562,E2 -28225.562} C_VEL
LIN {X 0,Y 107.281,Z 360.183,A -85,B 0,C 180,E1 -28226.658,E2 -28226.658} C_VEL
LIN {X 0,Y 110.36,Z 329.507,A -85,B 0,C 180,E1 -28228.342,E2 -28228.342} C_VEL
LIN {X 0,Y 107.103,Z 318.245,A -85,B 0,C 180,E1 -28231.468,E2 -28231.468} C_VEL
LIN {X 0,Y 104.054,Z 309.718,A -85,B 0,C 180,E1 -28234.475,E2 -28234.475} C_VEL
LIN {X 0,Y 100.01,Z 301.982,A -85,B 0,C 180,E1 -28238.533,E2 -28238.533} C_VEL
LIN {X 0,Y 95.593,Z 294.584,A -85,B 0,C 180,E1 -28243.757,E2 -28243.757} C_VEL
LIN {X 0,Y 93.301,Z 292.138,A -85,B 0,C 180,E1 -28246.701,E2 -28246.701} C_VEL
LIN {X 0,Y 90.972,Z 290.685,A -85,B 0,C 180,E1 -28249.975,E2 -28249.975} C_VEL
LIN {X 0,Y 85.751,Z 288.461,A -85,B 0,C 180,E1 -28259.746,E2 -28259.746} C_VEL
LIN {X 0,Y 84.901,Z 287.562,A -85,B 0,C 180,E1 -28262.32,E2 -28262.32} C_VEL
LIN {X 0,Y 83.422,Z 284.589,A -85,B 0,C 180,E1 -28269.672,E2 -28269.672} C_VEL
LIN {X 0,Y 83.123,Z 284.802,A -85,B 0,C 180,E1 -28282.168,E2 -28282.168} C_VEL
LIN {X 0,Y 84.127,Z 287.746,A -85,B 0,C 180,E1 -28288.987,E2 -28288.987} C_VEL
LIN {X 0,Y 86.254,Z 290.061,A -85,B 0,C 180,E1 -28295.612,E2 -28295.612} C_VEL
LIN {X 0,Y 88.528,Z 293.657,A -85,B 0,C 180,E1 -28300.76,E2 -28300.76} C_VEL
LIN {X 0,Y 89.604,Z 295.31,A -85,B 0,C 180,E1 -28302.781,E2 -28302.781} C_VEL
LIN {X 0,Y 92.159,Z 299.33,A -85,B 0,C 180,E1 -28307.006,E2 -28307.006} C_VEL
LIN {X 0,Y 95.596,Z 305.06,A -85,B 0,C 180,E1 -28311.655,E2 -28311.655} C_VEL
LIN {X 0,Y 99.009,Z 311.41,A -85,B 0,C 180,E1 -28315.657,E2 -28315.657} C_VEL
LIN {X 0,Y 104.136,Z 322.245,A -85,B 0,C 180,E1 -28320.805,E2 -28320.805} C_VEL
LIN {X 0,Y 105.7,Z 326.281,A -85,B 0,C 180,E1 -28322.262,E2 -28322.262} C_VEL
LIN {X 0,Y 102.139,Z 357.802,A -85,B 0,C 180,E1 -28323.963,E2 -28323.963} C_VEL
LIN {X 0,Y 99.646,Z 370.978,A -85,B 0,C 180,E1 -28325.244,E2 -28325.244} C_VEL
LIN {X 0,Y 96.529,Z 382.776,A -85,B 0,C 180,E1 -28326.963,E2 -28326.963} C_VEL
LIN {X 0,Y 92.405,Z 394.701,A -85,B 0,C 180,E1 -28329.405,E2 -28329.405} C_VEL
LIN {X 0,Y 87.392,Z 406.535,A -85,B 0,C 180,E1 -28332.816,E2 -28332.816} C_VEL
LIN {X 0,Y 82.095,Z 417.069,A -85,B 0,C 180,E1 -28337.014,E2 -28337.014} C_VEL
LIN {X 0,Y 76.742,Z 426.632,A -85,B 0,C 180,E1 -28342.406,E2 -28342.406} C_VEL
LIN {X 0,Y 72.037,Z 434.588,A -85,B 0,C 180,E1 -28348.602,E2 -28348.602} C_VEL
LIN {X 0,Y 68.033,Z 441.467,A -85,B 0,C 180,E1 -28355.929,E2 -28355.929} C_VEL
LIN {X 0,Y 65.096,Z 446.98,A -85,B 0,C 180,E1 -28363.833,E2 -28363.833} C_VEL
LIN {X 0,Y 63.094,Z 451.642,A -85,B 0,C 180,E1 -28372.712,E2 -28372.712} C_VEL
LIN {X 0,Y 62.181,Z 456.105,A -85,B 0,C 180,E1 -28384.409,E2 -28384.409} C_VEL
LIN {X 0,Y 62.824,Z 458.219,A -85,B 0,C 180,E1 -28392.159,E2 -28392.159} C_VEL
LIN {X 0,Y 64.525,Z 459.797,A -85,B 0,C 180,E1 -28399.677,E2 -28399.677} C_VEL
LIN {X 0,Y 68.267,Z 460.986,A -85,B 0,C 180,E1 -28409.061,E2 -28409.061} C_VEL
LIN {X 0,Y 75.113,Z 461.047,A -85,B 0,C 180,E1 -28419.329,E2 -28419.329} C_VEL
LIN {X 0,Y 80.499,Z 460.297,A -85,B 0,C 180,E1 -28424.846,E2 -28424.846} C_VEL
LIN {X 0,Y 88.303,Z 458.358,A -85,B 0,C 180,E1 -28430.867,E2 -28430.867} C_VEL
LIN {X 0,Y 98.557,Z 454.603,A -85,B 0,C 180,E1 -28436.649,E2 -28436.649} C_VEL
LIN {X 0,Y 109.104,Z 449.491,A -85,B 0,C 180,E1 -28441.087,E2 -28441.087} C_VEL
LIN {X 0,Y 117.704,Z 444.283,A -85,B 0,C 180,E1 -28443.949,E2 -28443.949} C_VEL
LIN {X 0,Y 127.356,Z 437.195,A -85,B 0,C 180,E1 -28446.645,E2 -28446.645} C_VEL
LIN {X 0,Y 137.016,Z 428.529,A -85,B 0,C 180,E1 -28448.868,E2 -28448.868} C_VEL
LIN {X 0,Y 145.886,Z 418.918,A -85,B 0,C 180,E1 -28450.615,E2 -28450.615} C_VEL
LIN {X 0,Y 153.559,Z 408.685,A -85,B 0,C 180,E1 -28451.972,E2 -28451.972} C_VEL
LIN {X 0,Y 160.126,Z 397.944,A -85,B 0,C 180,E1 -28452.98,E2 -28452.98} C_VEL
LIN {X 0,Y 166.04,Z 385.743,A -85,B 0,C 180,E1 -28453.874,E2 -28453.874} C_VEL
LIN {X 0,Y 169.678,Z 376,A -85,B 0,C 180,E1 -28454.403,E2 -28454.403} C_VEL
LIN {X 0,Y 169.824,Z 375.462,A -85,B 0,C 180,E1 -28456.852,E2 -28456.852} C_VEL
LIN {X 0,Y 169.905,Z 375.577,A -85,B 0,C 180,E1 -28457.945,E2 -28457.945} C_VEL
LIN {X 0,Y 166.507,Z 384.899,A -85,B 0,C 180,E1 -28458.404,E2 -28458.404} C_VEL
LIN {X 0,Y 160.768,Z 397.191,A -85,B 0,C 180,E1 -28459.036,E2 -28459.036} C_VEL
LIN {X 0,Y 154.139,Z 408.339,A -85,B 0,C 180,E1 -28459.886,E2 -28459.886} C_VEL
LIN {X 0,Y 145.949,Z 419.514,A -85,B 0,C 180,E1 -28461.101,E2 -28461.101} C_VEL
LIN {X 0,Y 137.048,Z 429.373,A -85,B 0,C 180,E1 -28462.626,E2 -28462.626} C_VEL
LIN {X 0,Y 127.528,Z 438.127,A -85,B 0,C 180,E1 -28464.594,E2 -28464.594} C_VEL
LIN {X 0,Y 118.206,Z 445.249,A -85,B 0,C 180,E1 -28466.899,E2 -28466.899} C_VEL
LIN {X 0,Y 109.276,Z 450.994,A -85,B 0,C 180,E1 -28469.748,E2 -28469.748} C_VEL
LIN {X 0,Y 100.584,Z 455.609,A -85,B 0,C 180,E1 -28473.025,E2 -28473.025} C_VEL
LIN {X 0,Y 92.49,Z 459.195,A -85,B 0,C 180,E1 -28477.076,E2 -28477.076} C_VEL
LIN {X 0,Y 84.953,Z 461.871,A -85,B 0,C 180,E1 -28481.881,E2 -28481.881} C_VEL
LIN {X 0,Y 76.009,Z 464.117,A -85,B 0,C 180,E1 -28489.668,E2 -28489.668} C_VEL
LIN {X 0,Y 68.94,Z 464.844,A -85,B 0,C 180,E1 -28499.356,E2 -28499.356} C_VEL
LIN {X 0,Y 64.516,Z 464.135,A -85,B 0,C 180,E1 -28510.926,E2 -28510.926} C_VEL
LIN {X 0,Y 62.847,Z 461.94,A -85,B 0,C 180,E1 -28523.58,E2 -28523.58} C_VEL
LIN {X 0,Y 62.928,Z 460.198,A -85,B 0,C 180,E1 -28530,E2 -28530} C_VEL
LIN {X 0,Y 63.074,Z 456.634,A -85,B 0,C 180,E1 -28539.622,E2 -28539.622} C_VEL
LIN {X 0,Y 64.548,Z 451.894,A -85,B 0,C 180,E1 -28549.065,E2 -28549.065} C_VEL
LIN {X 0,Y 68.191,Z 444.731,A -85,B 0,C 180,E1 -28559.311,E2 -28559.311} C_VEL
LIN {X 0,Y 72.803,Z 436.875,A -85,B 0,C 180,E1 -28567.109,E2 -28567.109} C_VEL
LIN {X 0,Y 78.168,Z 427.716,A -85,B 0,C 180,E1 -28573.497,E2 -28573.497} C_VEL
LIN {X 0,Y 83.402,Z 418.041,A -85,B 0,C 180,E1 -28578.313,E2 -28578.313} C_VEL
LIN {X 0,Y 88.204,Z 408.06,A -85,B 0,C 180,E1 -28581.889,E2 -28581.889} C_VEL
LIN {X 0,Y 92.669,Z 397.42,A -85,B 0,C 180,E1 -28584.613,E2 -28584.613} C_VEL
LIN {X 0,Y 96.999,Z 384.756,A -85,B 0,C 180,E1 -28586.902,E2 -28586.902} C_VEL
LIN {X 0,Y 100.287,Z 371.756,A -85,B 0,C 180,E1 -28588.517,E2 -28588.517} C_VEL
LIN {X 0,Y 102.507,Z 358.727,A -85,B 0,C 180,E1 -28589.511,E2 -28589.511} C_VEL
LIN {X 0,Y 105.424,Z 331.444,A -85,B 0,C 180,E1 -28590.966,E2 -28590.966} C_VEL
LIN {X 0,Y 102.268,Z 320.213,A -85,B 0,C 180,E1 -28594.385,E2 -28594.385} C_VEL
LIN {X 0,Y 100.165,Z 314.193,A -85,B 0,C 180,E1 -28596.711,E2 -28596.711} C_VEL
LIN {X 0,Y 96.618,Z 307.035,A -85,B 0,C 180,E1 -28600.745,E2 -28600.745} C_VEL
LIN {X 0,Y 92.819,Z 300.279,A -85,B 0,C 180,E1 -28605.729,E2 -28605.729} C_VEL
LIN {X 0,Y 90.973,Z 297.175,A -85,B 0,C 180,E1 -28608.572,E2 -28608.572} C_VEL
LIN {X 0,Y 88.642,Z 293.188,A -85,B 0,C 180,E1 -28612.88,E2 -28612.88} C_VEL
LIN {X 0,Y 86.601,Z 289.77,A -85,B 0,C 180,E1 -28617.43,E2 -28617.43} C_VEL
LIN {X 0,Y 84.901,Z 287.562,A -85,B 0,C 180,E1 -28622.32,E2 -28622.32} C_VEL
LIN {X 0,Y 83.861,Z 286.787,A -85,B 0,C 180,E1 -28626.233,E2 -28626.233} C_VEL
LIN {X 0,Y 82.966,Z 287.3,A -85,B 0,C 180,E1 -28630.262,E2 -28630.262} C_VEL
LIN {X 0,Y 82.197,Z 289.265,A -85,B 0,C 180,E1 -28635.681,E2 -28635.681} C_VEL
LIN {X 0,Y 82.188,Z 293.012,A -85,B 0,C 180,E1 -28643.874,E2 -28643.874} C_VEL
LIN {X 0,Y 84.664,Z 296.764,A -85,B 0,C 180,E1 -28654.269,E2 -28654.269} C_VEL
LIN {X 0,Y 87.3,Z 301.185,A -85,B 0,C 180,E1 -28660.651,E2 -28660.651} C_VEL
LIN {X 0,Y 89.754,Z 305.37,A -85,B 0,C 180,E1 -28665.194,E2 -28665.194} C_VEL
LIN {X 0,Y 92.862,Z 311.023,A -85,B 0,C 180,E1 -28669.917,E2 -28669.917} C_VEL
LIN {X 0,Y 95.628,Z 316.385,A -85,B 0,C 180,E1 -28673.461,E2 -28673.461} C_VEL
LIN {X 0,Y 100.266,Z 326.955,A -85,B 0,C 180,E1 -28678.75,E2 -28678.75} C_VEL
LIN {X 0,Y 100.86,Z 328.597,A -85,B 0,C 180,E1 -28679.386,E2 -28679.386} C_VEL
LIN {X 0,Y 97.338,Z 358.109,A -85,B 0,C 180,E1 -28680.945,E2 -28680.945} C_VEL
LIN {X 0,Y 94.818,Z 370.915,A -85,B 0,C 180,E1 -28682.174,E2 -28682.174} C_VEL
LIN {X 0,Y 91.321,Z 383.63,A -85,B 0,C 180,E1 -28684.043,E2 -28684.043} C_VEL
LIN {X 0,Y 86.627,Z 396.265,A -85,B 0,C 180,E1 -28686.7,E2 -28686.7} C_VEL
LIN {X 0,Y 81.748,Z 407.03,A -85,B 0,C 180,E1 -28689.886,E2 -28689.886} C_VEL
LIN {X 0,Y 76.356,Z 417.097,A -85,B 0,C 180,E1 -28693.971,E2 -28693.971} C_VEL
LIN {X 0,Y 70.336,Z 427.193,A -85,B 0,C 180,E1 -28699.929,E2 -28699.929} C_VEL
LIN {X 0,Y 65.069,Z 435.458,A -85,B 0,C 180,E1 -28706.904,E2 -28706.904} C_VEL
LIN {X 0,Y 60.835,Z 442.238,A -85,B 0,C 180,E1 -28714.968,E2 -28714.968} C_VEL
LIN {X 0,Y 57.742,Z 447.809,A -85,B 0,C 180,E1 -28724.088,E2 -28724.088} C_VEL
LIN {X 0,Y 55.651,Z 452.598,A -85,B 0,C 180,E1 -28734.734,E2 -28734.734} C_VEL
LIN {X 0,Y 55.112,Z 455.994,A -85,B 0,C 180,E1 -28745.018,E2 -28745.018} C_VEL
LIN {X 0,Y 56.742,Z 459.128,A -85,B 0,C 180,E1 -28757.999,E2 -28757.999} C_VEL
LIN {X 0,Y 59.27,Z 460.46,A -85,B 0,C 180,E1 -28766.099,E2 -28766.099} C_VEL
LIN {X 0,Y 62.819,Z 461.279,A -85,B 0,C 180,E1 -28773.506,E2 -28773.506} C_VEL
LIN {X 0,Y 69.043,Z 461.457,A -85,B 0,C 180,E1 -28782.255,E2 -28782.255} C_VEL
LIN {X 0,Y 78.318,Z 460.24,A -85,B 0,C 180,E1 -28790.778,E2 -28790.778} C_VEL
LIN {X 0,Y 85.109,Z 458.648,A -85,B 0,C 180,E1 -28795.29,E2 -28795.29} C_VEL
LIN {X 0,Y 94.415,Z 455.571,A -85,B 0,C 180,E1 -28800.024,E2 -28800.024} C_VEL
LIN {X 0,Y 105.722,Z 450.514,A -85,B 0,C 180,E1 -28804.357,E2 -28804.357} C_VEL
LIN {X 0,Y 114.679,Z 445.461,A -85,B 0,C 180,E1 -28807.06,E2 -28807.06} C_VEL
LIN {X 0,Y 123.093,Z 439.791,A -85,B 0,C 180,E1 -28809.2,E2 -28809.2} C_VEL
LIN {X 0,Y 132.54,Z 432.165,A -85,B 0,C 180,E1 -28811.204,E2 -28811.204} C_VEL
LIN {X 0,Y 141.445,Z 423.48,A -85,B 0,C 180,E1 -28812.818,E2 -28812.818} C_VEL
LIN {X 0,Y 149.982,Z 413.255,A -85,B 0,C 180,E1 -28814.195,E2 -28814.195} C_VEL
LIN {X 0,Y 157.744,Z 401.757,A -85,B 0,C 180,E1 -28815.27,E2 -28815.27} C_VEL
LIN {X 0,Y 161.686,Z 394.675,A -85,B 0,C 180,E1 -28815.8,E2 -28815.8} C_VEL
LIN {X 0,Y 161.18,Z 395.741,A -85,B 0,C 180,E1 -28816.414,E2 -28816.414} C_VEL
LIN {X 0,Y 154.436,Z 407.143,A -85,B 0,C 180,E1 -28817.132,E2 -28817.132} C_VEL
LIN {X 0,Y 146.081,Z 418.487,A -85,B 0,C 180,E1 -28818.168,E2 -28818.168} C_VEL
LIN {X 0,Y 137.798,Z 427.701,A -85,B 0,C 180,E1 -28819.35,E2 -28819.35} C_VEL
LIN {X 0,Y 128.009,Z 436.662,A -85,B 0,C 180,E1 -28821.043,E2 -28821.043} C_VEL
LIN {X 0,Y 116.727,Z 445.068,A -85,B 0,C 180,E1 -28823.342,E2 -28823.342} C_VEL
LIN {X 0,Y 109.022,Z 449.89,A -85,B 0,C 180,E1 -28825.516,E2 -28825.516} C_VEL
LIN {X 0,Y 99.886,Z 454.676,A -85,B 0,C 180,E1 -28828.421,E2 -28828.421} C_VEL
LIN {X 0,Y 91.174,Z 458.417,A -85,B 0,C 180,E1 -28832.017,E2 -28832.017} C_VEL
LIN {X 0,Y 80.375,Z 461.971,A -85,B 0,C 180,E1 -28838.1,E2 -28838.1} C_VEL
LIN {X 0,Y 70.731,Z 463.992,A -85,B 0,C 180,E1 -28845.932,E2 -28845.932} C_VEL
LIN {X 0,Y 62.921,Z 464.54,A -85,B 0,C 180,E1 -28856.051,E2 -28856.051} C_VEL
LIN {X 0,Y 57.835,Z 463.677,A -85,B 0,C 180,E1 -28868.621,E2 -28868.621} C_VEL
LIN {X 0,Y 55.827,Z 461.269,A -85,B 0,C 180,E1 -28882.769,E2 -28882.769} C_VEL
LIN {X 0,Y 55.858,Z 459.448,A -85,B 0,C 180,E1 -28890,E2 -28890} C_VEL
LIN {X 0,Y 56.093,Z 455.717,A -85,B 0,C 180,E1 -28900.833,E2 -28900.833} C_VEL
LIN {X 0,Y 57.858,Z 450.796,A -85,B 0,C 180,E1 -28911.371,E2 -28911.371} C_VEL
LIN {X 0,Y 61.35,Z 444.565,A -85,B 0,C 180,E1 -28921.03,E2 -28921.03} C_VEL
LIN {X 0,Y 66.305,Z 436.742,A -85,B 0,C 180,E1 -28929.491,E2 -28929.491} C_VEL
LIN {X 0,Y 72.103,Z 427.533,A -85,B 0,C 180,E1 -28936.297,E2 -28936.297} C_VEL
LIN {X 0,Y 77.68,Z 417.861,A -85,B 0,C 180,E1 -28941.29,E2 -28941.29} C_VEL
LIN {X 0,Y 82.692,Z 408.055,A -85,B 0,C 180,E1 -28944.886,E2 -28944.886} C_VEL
LIN {X 0,Y 87.375,Z 397.501,A -85,B 0,C 180,E1 -28947.624,E2 -28947.624} C_VEL
LIN {X 0,Y 91.906,Z 384.966,A -85,B 0,C 180,E1 -28949.888,E2 -28949.888} C_VEL
LIN {X 0,Y 95.43,Z 371.743,A -85,B 0,C 180,E1 -28951.537,E2 -28951.537} C_VEL
LIN {X 0,Y 97.815,Z 358.248,A -85,B 0,C 180,E1 -28952.552,E2 -28952.552} C_VEL
LIN {X 0,Y 100.569,Z 332.943,A -85,B 0,C 180,E1 -28953.941,E2 -28953.941} C_VEL
LIN {X 0,Y 97.765,Z 322.62,A -85,B 0,C 180,E1 -28957.43,E2 -28957.43} C_VEL
LIN {X 0,Y 96.508,Z 318.809,A -85,B 0,C 180,E1 -28959.042,E2 -28959.042} C_VEL
LIN {X 0,Y 93.612,Z 312.536,A -85,B 0,C 180,E1 -28962.752,E2 -28962.752} C_VEL
LIN {X 0,Y 89.939,Z 305.516,A -85,B 0,C 180,E1 -28968.199,E2 -28968.199} C_VEL
LIN {X 0,Y 88.279,Z 302.574,A -85,B 0,C 180,E1 -28971.171,E2 -28971.171} C_VEL
LIN {X 0,Y 86.462,Z 299.272,A -85,B 0,C 180,E1 -28974.964,E2 -28974.964} C_VEL
LIN {X 0,Y 84.568,Z 295.795,A -85,B 0,C 180,E1 -28979.973,E2 -28979.973} C_VEL
LIN {X 0,Y 82.374,Z 291.74,A -85,B 0,C 180,E1 -28989.796,E2 -28989.796} C_VEL
LIN {X 0,Y 81.943,Z 291.673,A -85,B 0,C 180,E1 -29000.033,E2 -29000.033} C_VEL
LIN {X 0,Y 82.059,Z 292.253,A -85,B 0,C 180,E1 -29002.186,E2 -29002.186} C_VEL
LIN {X 0,Y 82.188,Z 293.012,A -85,B 0,C 180,E1 -29003.874,E2 -29003.874} C_VEL
LIN {X 0,Y 82.664,Z 295.287,A -85,B 0,C 180,E1 -29007.66,E2 -29007.66} C_VEL
LIN {X 0,Y 83.652,Z 300.901,A -85,B 0,C 180,E1 -29013.274,E2 -29013.274} C_VEL
LIN {X 0,Y 85.664,Z 308.118,A -85,B 0,C 180,E1 -29019.693,E2 -29019.693} C_VEL
LIN {X 0,Y 86.736,Z 310.065,A -85,B 0,C 180,E1 -29021.914,E2 -29021.914} C_VEL
LIN {X 0,Y 89.719,Z 315.829,A -85,B 0,C 180,E1 -29027.261,E2 -29027.261} C_VEL
LIN {X 0,Y 92.813,Z 322.538,A -85,B 0,C 180,E1 -29031.811,E2 -29031.811} C_VEL
LIN {X 0,Y 96.315,Z 331.233,A -85,B 0,C 180,E1 -29036.292,E2 -29036.292} C_VEL
LIN {X 0,Y 92.899,Z 358.11,A -85,B 0,C 180,E1 -29037.612,E2 -29037.612} C_VEL
LIN {X 0,Y 90.284,Z 370.922,A -85,B 0,C 180,E1 -29038.801,E2 -29038.801} C_VEL
LIN {X 0,Y 86.911,Z 382.727,A -85,B 0,C 180,E1 -29040.457,E2 -29040.457} C_VEL
LIN {X 0,Y 82.502,Z 394.455,A -85,B 0,C 180,E1 -29042.75,E2 -29042.75} C_VEL
LIN {X 0,Y 76.732,Z 406.743,A -85,B 0,C 180,E1 -29046.255,E2 -29046.255} C_VEL
LIN {X 0,Y 70.897,Z 417.104,A -85,B 0,C 180,E1 -29050.454,E2 -29050.454} C_VEL
LIN {X 0,Y 64.813,Z 426.674,A -85,B 0,C 180,E1 -29056.169,E2 -29056.169} C_VEL
LIN {X 0,Y 59.219,Z 434.779,A -85,B 0,C 180,E1 -29063.184,E2 -29063.184} C_VEL
LIN {X 0,Y 54.482,Z 441.704,A -85,B 0,C 180,E1 -29071.848,E2 -29071.848} C_VEL
LIN {X 0,Y 50.559,Z 448.18,A -85,B 0,C 180,E1 -29083.542,E2 -29083.542} C_VEL
LIN {X 0,Y 48.397,Z 452.96,A -85,B 0,C 180,E1 -29095.825,E2 -29095.825} C_VEL
LIN {X 0,Y 48.034,Z 455.86,A -85,B 0,C 180,E1 -29105.819,E2 -29105.819} C_VEL
LIN {X 0,Y 49.031,Z 458.206,A -85,B 0,C 180,E1 -29115.779,E2 -29115.779} C_VEL
LIN {X 0,Y 52.174,Z 460.285,A -85,B 0,C 180,E1 -29127.451,E2 -29127.451} C_VEL
LIN {X 0,Y 57.727,Z 461.56,A -85,B 0,C 180,E1 -29138.622,E2 -29138.622} C_VEL
LIN {X 0,Y 64.91,Z 461.744,A -85,B 0,C 180,E1 -29147.53,E2 -29147.53} C_VEL
LIN {X 0,Y 73.291,Z 460.873,A -85,B 0,C 180,E1 -29154.529,E2 -29154.529} C_VEL
LIN {X 0,Y 84.344,Z 458.419,A -85,B 0,C 180,E1 -29160.918,E2 -29160.918} C_VEL
LIN {X 0,Y 95.444,Z 454.689,A -85,B 0,C 180,E1 -29165.504,E2 -29165.504} C_VEL
LIN {X 0,Y 106.717,Z 449.607,A -85,B 0,C 180,E1 -29168.955,E2 -29168.955} C_VEL
LIN {X 0,Y 116.487,Z 444.004,A -85,B 0,C 180,E1 -29171.369,E2 -29171.369} C_VEL
LIN {X 0,Y 127.121,Z 436.471,A -85,B 0,C 180,E1 -29173.507,E2 -29173.507} C_VEL
LIN {X 0,Y 136.803,Z 428.071,A -85,B 0,C 180,E1 -29175.098,E2 -29175.098} C_VEL
LIN {X 0,Y 138.471,Z 426.425,A -85,B 0,C 180,E1 -29175.356,E2 -29175.356} C_VEL
LIN {X 0,Y 139.01,Z 425.928,A -85,B 0,C 180,E1 -29176.144,E2 -29176.144} C_VEL
LIN {X 0,Y 128.979,Z 435.244,A -85,B 0,C 180,E1 -29177.534,E2 -29177.534} C_VEL
LIN {X 0,Y 119.057,Z 442.751,A -85,B 0,C 180,E1 -29179.185,E2 -29179.185} C_VEL
LIN {X 0,Y 112.545,Z 446.947,A -85,B 0,C 180,E1 -29180.502,E2 -29180.502} C_VEL
LIN {X 0,Y 103.007,Z 452.223,A -85,B 0,C 180,E1 -29182.919,E2 -29182.919} C_VEL
LIN {X 0,Y 93.622,Z 456.443,A -85,B 0,C 180,E1 -29185.738,E2 -29185.738} C_VEL
LIN {X 0,Y 81.805,Z 460.591,A -85,B 0,C 180,E1 -29190.786,E2 -29190.786} C_VEL
LIN {X 0,Y 70.856,Z 463.129,A -85,B 0,C 180,E1 -29197.489,E2 -29197.489} C_VEL
LIN {X 0,Y 61.246,Z 464.222,A -85,B 0,C 180,E1 -29206.491,E2 -29206.491} C_VEL
LIN {X 0,Y 53.803,Z 463.881,A -85,B 0,C 180,E1 -29218.501,E2 -29218.501} C_VEL
LIN {X 0,Y 49.573,Z 462.047,A -85,B 0,C 180,E1 -29233.529,E2 -29233.529} C_VEL
LIN {X 0,Y 48.829,Z 460.574,A -85,B 0,C 180,E1 -29241.725,E2 -29241.725} C_VEL
LIN {X 0,Y 48.784,Z 458.68,A -85,B 0,C 180,E1 -29250.001,E2 -29250.001} C_VEL
LIN {X 0,Y 49.136,Z 454.788,A -85,B 0,C 180,E1 -29262.389,E2 -29262.389} C_VEL
LIN {X 0,Y 51.86,Z 448.694,A -85,B 0,C 180,E1 -29276.131,E2 -29276.131} C_VEL
LIN {X 0,Y 56.198,Z 441.975,A -85,B 0,C 180,E1 -29286.443,E2 -29286.443} C_VEL
LIN {X 0,Y 62.013,Z 433.605,A -85,B 0,C 180,E1 -29295.098,E2 -29295.098} C_VEL
LIN {X 0,Y 68.3,Z 424.099,A -85,B 0,C 180,E1 -29301.553,E2 -29301.553} C_VEL
LIN {X 0,Y 74.056,Z 414.305,A -85,B 0,C 180,E1 -29306.137,E2 -29306.137} C_VEL
LIN {X 0,Y 79.545,Z 403.821,A -85,B 0,C 180,E1 -29309.476,E2 -29309.476} C_VEL
LIN {X 0,Y 84.509,Z 392.22,A -85,B 0,C 180,E1 -29312.078,E2 -29312.078} C_VEL
LIN {X 0,Y 88.546,Z 380.379,A -85,B 0,C 180,E1 -29313.879,E2 -29313.879} C_VEL
LIN {X 0,Y 91.888,Z 366.939,A -85,B 0,C 180,E1 -29315.263,E2 -29315.263} C_VEL
LIN {X 0,Y 93.958,Z 353.102,A -85,B 0,C 180,E1 -29316.138,E2 -29316.138} C_VEL
LIN {X 0,Y 95.977,Z 334.68,A -85,B 0,C 180,E1 -29317.154,E2 -29317.154} C_VEL
LIN {X 0,Y 93.535,Z 324.933,A -85,B 0,C 180,E1 -29320.802,E2 -29320.802} C_VEL
LIN {X 0,Y 91.271,Z 319.248,A -85,B 0,C 180,E1 -29324.019,E2 -29324.019} C_VEL
LIN {X 0,Y 87.998,Z 312.346,A -85,B 0,C 180,E1 -29329.362,E2 -29329.362} C_VEL
LIN {X 0,Y 86.072,Z 308.619,A -85,B 0,C 180,E1 -29333.192,E2 -29333.192} C_VEL
LIN {X 0,Y 84.446,Z 305.391,A -85,B 0,C 180,E1 -29337.047,E2 -29337.047} C_VEL
LIN {X 0,Y 83.008,Z 302.416,A -85,B 0,C 180,E1 -29341.506,E2 -29341.506} C_VEL
LIN {X 0,Y 81.219,Z 298.732,A -85,B 0,C 180,E1 -29350.793,E2 -29350.793} C_VEL
LIN {X 0,Y 80.952,Z 298.734,A -85,B 0,C 180,E1 -29360.289,E2 -29360.289} C_VEL
LIN {X 0,Y 82.05,Z 302.102,A -85,B 0,C 180,E1 -29369.031,E2 -29369.031} C_VEL
LIN {X 0,Y 83.186,Z 303.59,A -85,B 0,C 180,E1 -29373.093,E2 -29373.093} C_VEL
LIN {X 0,Y 85.343,Z 307.576,A -85,B 0,C 180,E1 -29378.99,E2 -29378.99} C_VEL
LIN {X 0,Y 86.736,Z 310.065,A -85,B 0,C 180,E1 -29381.914,E2 -29381.914} C_VEL
LIN {X 0,Y 87.672,Z 312.455,A -85,B 0,C 180,E1 -29383.827,E2 -29383.827} C_VEL
LIN {X 0,Y 88.207,Z 315.713,A -85,B 0,C 180,E1 -29385.264,E2 -29385.264} C_VEL
LIN {X 0,Y 89.128,Z 325.526,A -85,B 0,C 180,E1 -29388.42,E2 -29388.42} C_VEL
LIN {X 0,Y 89.674,Z 327.695,A -85,B 0,C 180,E1 -29389.447,E2 -29389.447} C_VEL
LIN {X 0,Y 91.974,Z 333.722,A -85,B 0,C 180,E1 -29392.829,E2 -29392.829} C_VEL
LIN {X 0,Y 88.618,Z 358.905,A -85,B 0,C 180,E1 -29394.033,E2 -29394.033} C_VEL
LIN {X 0,Y 85.856,Z 371.711,A -85,B 0,C 180,E1 -29395.204,E2 -29395.204} C_VEL
LIN {X 0,Y 82.022,Z 384.274,A -85,B 0,C 180,E1 -29396.952,E2 -29396.952} C_VEL
LIN {X 0,Y 77.296,Z 395.875,A -85,B 0,C 180,E1 -29399.24,E2 -29399.24} C_VEL
LIN {X 0,Y 71.129,Z 408.037,A -85,B 0,C 180,E1 -29402.703,E2 -29402.703} C_VEL
LIN {X 0,Y 64.294,Z 419.187,A -85,B 0,C 180,E1 -29407.506,E2 -29407.506} C_VEL
LIN {X 0,Y 57.745,Z 428.611,A -85,B 0,C 180,E1 -29413.701,E2 -29413.701} C_VEL
LIN {X 0,Y 51.397,Z 437.051,A -85,B 0,C 180,E1 -29422.14,E2 -29422.14} C_VEL
LIN {X 0,Y 46.499,Z 443.632,A -85,B 0,C 180,E1 -29432.165,E2 -29432.165} C_VEL
LIN {X 0,Y 42.674,Z 449.69,A -85,B 0,C 180,E1 -29445.935,E2 -29445.935} C_VEL
LIN {X 0,Y 40.943,Z 454.279,A -85,B 0,C 180,E1 -29460.993,E2 -29460.993} C_VEL
LIN {X 0,Y 42.244,Z 458.116,A -85,B 0,C 180,E1 -29478.357,E2 -29478.357} C_VEL
LIN {X 0,Y 46.958,Z 460.674,A -85,B 0,C 180,E1 -29493.891,E2 -29493.891} C_VEL
LIN {X 0,Y 53.292,Z 461.842,A -85,B 0,C 180,E1 -29504.752,E2 -29504.752} C_VEL
LIN {X 0,Y 61.407,Z 462.031,A -85,B 0,C 180,E1 -29513.466,E2 -29513.466} C_VEL
LIN {X 0,Y 70.583,Z 461.169,A -85,B 0,C 180,E1 -29520.032,E2 -29520.032} C_VEL
LIN {X 0,Y 80.534,Z 459.233,A -85,B 0,C 180,E1 -29525.035,E2 -29525.035} C_VEL
LIN {X 0,Y 92.61,Z 455.57,A -85,B 0,C 180,E1 -29529.419,E2 -29529.419} C_VEL
LIN {X 0,Y 101.93,Z 451.783,A -85,B 0,C 180,E1 -29531.96,E2 -29531.96} C_VEL
LIN {X 0,Y 113.106,Z 446,A -85,B 0,C 180,E1 -29534.411,E2 -29534.411} C_VEL
LIN {X 0,Y 116.446,Z 443.998,A -85,B 0,C 180,E1 -29535.064,E2 -29535.064} C_VEL
LIN {X 0,Y 116.932,Z 443.735,A -85,B 0,C 180,E1 -29535.924,E2 -29535.924} C_VEL
LIN {X 0,Y 107.015,Z 449.581,A -85,B 0,C 180,E1 -29537.781,E2 -29537.781} C_VEL
LIN {X 0,Y 97.215,Z 454.289,A -85,B 0,C 180,E1 -29539.985,E2 -29539.985} C_VEL
LIN {X 0,Y 87.621,Z 457.973,A -85,B 0,C 180,E1 -29542.724,E2 -29542.724} C_VEL
LIN {X 0,Y 74.067,Z 461.76,A -85,B 0,C 180,E1 -29548.356,E2 -29548.356} C_VEL
LIN {X 0,Y 66.764,Z 463.078,A -85,B 0,C 180,E1 -29552.637,E2 -29552.637} C_VEL
LIN {X 0,Y 56.305,Z 463.987,A -85,B 0,C 180,E1 -29561.506,E2 -29561.506} C_VEL
LIN {X 0,Y 47.872,Z 463.412,A -85,B 0,C 180,E1 -29574.041,E2 -29574.041} C_VEL
LIN {X 0,Y 42.819,Z 461.426,A -85,B 0,C 180,E1 -29590.838,E2 -29590.838} C_VEL
LIN {X 0,Y 41.636,Z 458.885,A -85,B 0,C 180,E1 -29605.159,E2 -29605.159} C_VEL
LIN {X 0,Y 41.729,Z 457.83,A -85,B 0,C 180,E1 -29610.001,E2 -29610.001} C_VEL
LIN {X 0,Y 42.236,Z 453.758,A -85,B 0,C 180,E1 -29624.454,E2 -29624.454} C_VEL
LIN {X 0,Y 45.579,Z 447.434,A -85,B 0,C 180,E1 -29640.075,E2 -29640.075} C_VEL
LIN {X 0,Y 50.646,Z 440.508,A -85,B 0,C 180,E1 -29651.234,E2 -29651.234} C_VEL
LIN {X 0,Y 57.208,Z 431.79,A -85,B 0,C 180,E1 -29660.157,E2 -29660.157} C_VEL
LIN {X 0,Y 63.507,Z 422.861,A -85,B 0,C 180,E1 -29666.079,E2 -29666.079} C_VEL
LIN {X 0,Y 69.616,Z 413.001,A -85,B 0,C 180,E1 -29670.541,E2 -29670.541} C_VEL
LIN {X 0,Y 75.446,Z 402.283,A -85,B 0,C 180,E1 -29673.712,E2 -29673.712} C_VEL
LIN {X 0,Y 80.68,Z 390.325,A -85,B 0,C 180,E1 -29676.153,E2 -29676.153} C_VEL
LIN {X 0,Y 84.931,Z 377.821,A -85,B 0,C 180,E1 -29677.892,E2 -29677.892} C_VEL
LIN {X 0,Y 88.044,Z 364.956,A -85,B 0,C 180,E1 -29679.045,E2 -29679.045} C_VEL
LIN {X 0,Y 90.53,Z 347.518,A -85,B 0,C 180,E1 -29679.998,E2 -29679.998} C_VEL
LIN {X 0,Y 91.765,Z 336.729,A -85,B 0,C 180,E1 -29680.579,E2 -29680.579} C_VEL
LIN {X 0,Y 89.769,Z 328.329,A -85,B 0,C 180,E1 -29684.016,E2 -29684.016} C_VEL
LIN {X 0,Y 87.484,Z 322.581,A -85,B 0,C 180,E1 -29687.863,E2 -29687.863} C_VEL
LIN {X 0,Y 84.937,Z 316.637,A -85,B 0,C 180,E1 -29693.03,E2 -29693.03} C_VEL
LIN {X 0,Y 82.712,Z 311.825,A -85,B 0,C 180,E1 -29698.729,E2 -29698.729} C_VEL
LIN {X 0,Y 81.538,Z 309.044,A -85,B 0,C 180,E1 -29703.001,E2 -29703.001} C_VEL
LIN {X 0,Y 80.16,Z 305.787,A -85,B 0,C 180,E1 -29711.154,E2 -29711.154} C_VEL
LIN {X 0,Y 79.899,Z 305.738,A -85,B 0,C 180,E1 -29719.391,E2 -29719.391} C_VEL
LIN {X 0,Y 80.948,Z 309.178,A -85,B 0,C 180,E1 -29728.779,E2 -29728.779} C_VEL
LIN {X 0,Y 81.67,Z 310.262,A -85,B 0,C 180,E1 -29731.588,E2 -29731.588} C_VEL
LIN {X 0,Y 83.473,Z 313.957,A -85,B 0,C 180,E1 -29737.276,E2 -29737.276} C_VEL
LIN {X 0,Y 85.576,Z 318.248,A -85,B 0,C 180,E1 -29742.089,E2 -29742.089} C_VEL
LIN {X 0,Y 88.525,Z 324.765,A -85,B 0,C 180,E1 -29747.563,E2 -29747.563} C_VEL
LIN {X 0,Y 89.674,Z 327.695,A -85,B 0,C 180,E1 -29749.447,E2 -29749.447} C_VEL
LIN {X 0,Y 90.059,Z 330.447,A -85,B 0,C 180,E1 -29750.358,E2 -29750.358} C_VEL
LIN {X 0,Y 89.726,Z 334.282,A -85,B 0,C 180,E1 -29750.681,E2 -29750.681} C_VEL
LIN {X 0,Y 88.296,Z 340.304,A -85,B 0,C 180,E1 -29750.225,E2 -29750.225} C_VEL
LIN {X 0,Y 86.577,Z 347.301,A -85,B 0,C 180,E1 -29749.603,E2 -29749.603} C_VEL
LIN {X 0,Y 86.352,Z 348.732,A -85,B 0,C 180,E1 -29749.617,E2 -29749.617} C_VEL
LIN {X 0,Y 84.124,Z 362.457,A -85,B 0,C 180,E1 -29750.295,E2 -29750.295} C_VEL
LIN {X 0,Y 81.183,Z 374.574,A -85,B 0,C 180,E1 -29751.508,E2 -29751.508} C_VEL
LIN {X 0,Y 76.506,Z 387.91,A -85,B 0,C 180,E1 -29753.338,E2 -29753.338} C_VEL
LIN {X 0,Y 71.529,Z 398.982,A -85,B 0,C 180,E1 -29755.601,E2 -29755.601} C_VEL
LIN {X 0,Y 64.97,Z 410.683,A -85,B 0,C 180,E1 -29759.098,E2 -29759.098} C_VEL
LIN {X 0,Y 57.896,Z 421.238,A -85,B 0,C 180,E1 -29763.894,E2 -29763.894} C_VEL
LIN {X 0,Y 50.884,Z 430.383,A -85,B 0,C 180,E1 -29770.409,E2 -29770.409} C_VEL
LIN {X 0,Y 43.576,Z 439.17,A -85,B 0,C 180,E1 -29780.718,E2 -29780.718} C_VEL
LIN {X 0,Y 38.493,Z 445.438,A -85,B 0,C 180,E1 -29792.615,E2 -29792.615} C_VEL
LIN {X 0,Y 35.047,Z 450.683,A -85,B 0,C 180,E1 -29807.796,E2 -29807.796} C_VEL
LIN {X 0,Y 33.94,Z 455.546,A -85,B 0,C 180,E1 -29828.403,E2 -29828.403} C_VEL
LIN {X 0,Y 36.037,Z 458.394,A -85,B 0,C 180,E1 -29844.273,E2 -29844.273} C_VEL
LIN {X 0,Y 41.676,Z 460.84,A -85,B 0,C 180,E1 -29860.349,E2 -29860.349} C_VEL
LIN {X 0,Y 49.67,Z 462.137,A -85,B 0,C 180,E1 -29872.064,E2 -29872.064} C_VEL
LIN {X 0,Y 58.615,Z 462.321,A -85,B 0,C 180,E1 -29880.039,E2 -29880.039} C_VEL
LIN {X 0,Y 70.795,Z 461.14,A -85,B 0,C 180,E1 -29886.931,E2 -29886.931} C_VEL
LIN {X 0,Y 79.167,Z 459.556,A -85,B 0,C 180,E1 -29890.256,E2 -29890.256} C_VEL
LIN {X 0,Y 91.973,Z 455.839,A -85,B 0,C 180,E1 -29894.019,E2 -29894.019} C_VEL
LIN {X 0,Y 96.309,Z 454.248,A -85,B 0,C 180,E1 -29895.042,E2 -29895.042} C_VEL
LIN {X 0,Y 95.036,Z 454.821,A -85,B 0,C 180,E1 -29895.986,E2 -29895.986} C_VEL
LIN {X 0,Y 85.132,Z 458.31,A -85,B 0,C 180,E1 -29898.316,E2 -29898.316} C_VEL
LIN {X 0,Y 75.519,Z 460.875,A -85,B 0,C 180,E1 -29901.473,E2 -29901.473} C_VEL
LIN {X 0,Y 63.212,Z 463.023,A -85,B 0,C 180,E1 -29907.199,E2 -29907.199} C_VEL
LIN {X 0,Y 51.871,Z 463.683,A -85,B 0,C 180,E1 -29915.62,E2 -29915.62} C_VEL
LIN {X 0,Y 42.314,Z 462.936,A -85,B 0,C 180,E1 -29928.369,E2 -29928.369} C_VEL
LIN {X 0,Y 36.202,Z 460.761,A -85,B 0,C 180,E1 -29947.155,E2 -29947.155} C_VEL
LIN {X 0,Y 34.611,Z 458.096,A -85,B 0,C 180,E1 -29964.174,E2 -29964.174} C_VEL
LIN {X 0,Y 34.661,Z 456.958,A -85,B 0,C 180,E1 -29970.001,E2 -29970.001} C_VEL
LIN {X 0,Y 35.394,Z 452.696,A -85,B 0,C 180,E1 -29987.329,E2 -29987.329} C_VEL
LIN {X 0,Y 38.79,Z 447.188,A -85,B 0,C 180,E1 -30002.925,E2 -30002.925} C_VEL
LIN {X 0,Y 44.426,Z 440.266,A -85,B 0,C 180,E1 -30015.388,E2 -30015.388} C_VEL
LIN {X 0,Y 51.628,Z 431.561,A -85,B 0,C 180,E1 -30024.761,E2 -30024.761} C_VEL
LIN {X 0,Y 59.198,Z 421.546,A -85,B 0,C 180,E1 -30031.293,E2 -30031.293} C_VEL
LIN {X 0,Y 65.663,Z 411.574,A -85,B 0,C 180,E1 -30035.471,E2 -30035.471} C_VEL
LIN {X 0,Y 71.802,Z 400.515,A -85,B 0,C 180,E1 -30038.411,E2 -30038.411} C_VEL
LIN {X 0,Y 77.294,Z 388.202,A -85,B 0,C 180,E1 -30040.618,E2 -30040.618} C_VEL
LIN {X 0,Y 81.65,Z 375.109,A -85,B 0,C 180,E1 -30042.181,E2 -30042.181} C_VEL
LIN {X 0,Y 84.875,Z 361.143,A -85,B 0,C 180,E1 -30043.196,E2 -30043.196} C_VEL
LIN {X 0,Y 87.786,Z 338.588,A -85,B 0,C 180,E1 -30044.335,E2 -30044.335} C_VEL
LIN {X 0,Y 86.375,Z 332.251,A -85,B 0,C 180,E1 -30047.288,E2 -30047.288} C_VEL
LIN {X 0,Y 84.263,Z 326.378,A -85,B 0,C 180,E1 -30051.688,E2 -30051.688} C_VEL
LIN {X 0,Y 82.252,Z 321.351,A -85,B 0,C 180,E1 -30056.621,E2 -30056.621} C_VEL
LIN {X 0,Y 80.806,Z 317.686,A -85,B 0,C 180,E1 -30061.39,E2 -30061.39} C_VEL
LIN {X 0,Y 80.015,Z 315.49,A -85,B 0,C 180,E1 -30065.01,E2 -30065.01} C_VEL
LIN {X 0,Y 79.058,Z 312.733,A -85,B 0,C 180,E1 -30072.084,E2 -30072.084} C_VEL
LIN {X 0,Y 78.867,Z 312.793,A -85,B 0,C 180,E1 -30078.765,E2 -30078.765} C_VEL
LIN {X 0,Y 79.713,Z 316.064,A -85,B 0,C 180,E1 -30087.916,E2 -30087.916} C_VEL
LIN {X 0,Y 80.278,Z 317.087,A -85,B 0,C 180,E1 -30090.382,E2 -30090.382} C_VEL
LIN {X 0,Y 81.752,Z 320.592,A -85,B 0,C 180,E1 -30095.737,E2 -30095.737} C_VEL
LIN {X 0,Y 83.677,Z 324.928,A -85,B 0,C 180,E1 -30100.713,E2 -30100.713} C_VEL
LIN {X 0,Y 86.329,Z 331.741,A -85,B 0,C 180,E1 -30106.209,E2 -30106.209} C_VEL
LIN {X 0,Y 87.926,Z 336.41,A -85,B 0,C 180,E1 -30109.094,E2 -30109.094} C_VEL
LIN {X 0,Y 86.352,Z 348.732,A -85,B 0,C 180,E1 -30109.617,E2 -30109.617} C_VEL
LIN {X 0,Y 85.199,Z 354.516,A -85,B 0,C 180,E1 -30109.448,E2 -30109.448} C_VEL
LIN {X 0,Y 82.097,Z 363.772,A -85,B 0,C 180,E1 -30108.284,E2 -30108.284} C_VEL
LIN {X 0,Y 78.465,Z 372.882,A -85,B 0,C 180,E1 -30107.275,E2 -30107.275} C_VEL
LIN {X 0,Y 76.446,Z 378.436,A -85,B 0,C 180,E1 -30107.452,E2 -30107.452} C_VEL
LIN {X 0,Y 72.184,Z 389.539,A -85,B 0,C 180,E1 -30108.915,E2 -30108.915} C_VEL
LIN {X 0,Y 66.974,Z 400.282,A -85,B 0,C 180,E1 -30110.979,E2 -30110.979} C_VEL
LIN {X 0,Y 60.128,Z 411.711,A -85,B 0,C 180,E1 -30114.238,E2 -30114.238} C_VEL
LIN {X 0,Y 52.585,Z 422.152,A -85,B 0,C 180,E1 -30118.809,E2 -30118.809} C_VEL
LIN {X 0,Y 45.471,Z 430.653,A -85,B 0,C 180,E1 -30124.847,E2 -30124.847} C_VEL
LIN {X 0,Y 38.319,Z 438.436,A -85,B 0,C 180,E1 -30134.031,E2 -30134.031} C_VEL
LIN {X 0,Y 32.351,Z 444.869,A -85,B 0,C 180,E1 -30146.886,E2 -30146.886} C_VEL
LIN {X 0,Y 28.209,Z 450.188,A -85,B 0,C 180,E1 -30164.425,E2 -30164.425} C_VEL
LIN {X 0,Y 26.837,Z 454.91,A -85,B 0,C 180,E1 -30188.363,E2 -30188.363} C_VEL
LIN {X 0,Y 31.049,Z 459.04,A -85,B 0,C 180,E1 -30214.875,E2 -30214.875} C_VEL
LIN {X 0,Y 37.525,Z 461.104,A -85,B 0,C 180,E1 -30229.268,E2 -30229.268} C_VEL
LIN {X 0,Y 46.607,Z 462.39,A -85,B 0,C 180,E1 -30240.049,E2 -30240.049} C_VEL
LIN {X 0,Y 56.664,Z 462.612,A -85,B 0,C 180,E1 -30247.165,E2 -30247.165} C_VEL
LIN {X 0,Y 67.391,Z 461.781,A -85,B 0,C 180,E1 -30252.073,E2 -30252.073} C_VEL
LIN {X 0,Y 74.966,Z 460.576,A -85,B 0,C 180,E1 -30254.606,E2 -30254.606} C_VEL
LIN {X 0,Y 73.22,Z 461.014,A -85,B 0,C 180,E1 -30256.297,E2 -30256.297} C_VEL
LIN {X 0,Y 60.287,Z 462.898,A -85,B 0,C 180,E1 -30261.161,E2 -30261.161} C_VEL
LIN {X 0,Y 48.075,Z 463.376,A -85,B 0,C 180,E1 -30268.706,E2 -30268.706} C_VEL
LIN {X 0,Y 37.295,Z 462.443,A -85,B 0,C 180,E1 -30281.085,E2 -30281.085} C_VEL
LIN {X 0,Y 29.806,Z 460.027,A -85,B 0,C 180,E1 -30301.865,E2 -30301.865} C_VEL
LIN {X 0,Y 27.61,Z 457.2,A -85,B 0,C 180,E1 -30322.689,E2 -30322.689} C_VEL
LIN {X 0,Y 27.608,Z 456.046,A -85,B 0,C 180,E1 -30330.001,E2 -30330.001} C_VEL
LIN {X 0,Y 28.688,Z 451.598,A -85,B 0,C 180,E1 -30351.56,E2 -30351.56} C_VEL
LIN {X 0,Y 34.016,Z 444.759,A -85,B 0,C 180,E1 -30372.181,E2 -30372.181} C_VEL
LIN {X 0,Y 41.037,Z 437.31,A -85,B 0,C 180,E1 -30384.437,E2 -30384.437} C_VEL
LIN {X 0,Y 47.877,Z 429.689,A -85,B 0,C 180,E1 -30391.732,E2 -30391.732} C_VEL
LIN {X 0,Y 55.489,Z 420.106,A -85,B 0,C 180,E1 -30397.332,E2 -30397.332} C_VEL
LIN {X 0,Y 63.045,Z 408.792,A -85,B 0,C 180,E1 -30401.356,E2 -30401.356} C_VEL
LIN {X 0,Y 69.498,Z 397.144,A -85,B 0,C 180,E1 -30403.879,E2 -30403.879} C_VEL
LIN {X 0,Y 74.835,Z 384.842,A -85,B 0,C 180,E1 -30405.572,E2 -30405.572} C_VEL
LIN {X 0,Y 79.152,Z 371.259,A -85,B 0,C 180,E1 -30406.884,E2 -30406.884} C_VEL
LIN {X 0,Y 81.921,Z 358.005,A -85,B 0,C 180,E1 -30407.624,E2 -30407.624} C_VEL
LIN {X 0,Y 84.179,Z 340.638,A -85,B 0,C 180,E1 -30408.442,E2 -30408.442} C_VEL
LIN {X 0,Y 83.36,Z 336.53,A -85,B 0,C 180,E1 -30410.611,E2 -30410.611} C_VEL
LIN {X 0,Y 81.214,Z 329.925,A -85,B 0,C 180,E1 -30416.091,E2 -30416.091} C_VEL
LIN {X 0,Y 79.472,Z 324.693,A -85,B 0,C 180,E1 -30422.289,E2 -30422.289} C_VEL
LIN {X 0,Y 78.595,Z 322.005,A -85,B 0,C 180,E1 -30426.853,E2 -30426.853} C_VEL
LIN {X 0,Y 77.996,Z 319.721,A -85,B 0,C 180,E1 -30432.72,E2 -30432.72} C_VEL
LIN {X 0,Y 77.837,Z 319.883,A -85,B 0,C 180,E1 -30438.068,E2 -30438.068} C_VEL
LIN {X 0,Y 78.843,Z 323.744,A -85,B 0,C 180,E1 -30448.85,E2 -30448.85} C_VEL
LIN {X 0,Y 80.019,Z 326.922,A -85,B 0,C 180,E1 -30453.834,E2 -30453.834} C_VEL
LIN {X 0,Y 81.472,Z 330.771,A -85,B 0,C 180,E1 -30458.357,E2 -30458.357} C_VEL
LIN {X 0,Y 83.651,Z 337.08,A -85,B 0,C 180,E1 -30463.629,E2 -30463.629} C_VEL
LIN {X 0,Y 84.204,Z 338.994,A -85,B 0,C 180,E1 -30464.879,E2 -30464.879} C_VEL
LIN {X 0,Y 81.566,Z 358.265,A -85,B 0,C 180,E1 -30465.75,E2 -30465.75} C_VEL
LIN {X 0,Y 78.681,Z 370.999,A -85,B 0,C 180,E1 -30466.673,E2 -30466.673} C_VEL
LIN {X 0,Y 76.446,Z 378.436,A -85,B 0,C 180,E1 -30467.452,E2 -30467.452} C_VEL
LIN {X 0,Y 74.206,Z 383.901,A -85,B 0,C 180,E1 -30467.641,E2 -30467.641} C_VEL
LIN {X 0,Y 69.248,Z 392.441,A -85,B 0,C 180,E1 -30466.846,E2 -30466.846} C_VEL
LIN {X 0,Y 63.671,Z 400.64,A -85,B 0,C 180,E1 -30466.132,E2 -30466.132} C_VEL
LIN {X 0,Y 60.435,Z 405.577,A -85,B 0,C 180,E1 -30466.66,E2 -30466.66} C_VEL
LIN {X 0,Y 53.044,Z 416.327,A -85,B 0,C 180,E1 -30469.767,E2 -30469.767} C_VEL
LIN {X 0,Y 45.384,Z 425.715,A -85,B 0,C 180,E1 -30474.223,E2 -30474.223} C_VEL
LIN {X 0,Y 36.854,Z 434.648,A -85,B 0,C 180,E1 -30481.527,E2 -30481.527} C_VEL
LIN {X 0,Y 29.447,Z 441.697,A -85,B 0,C 180,E1 -30492.411,E2 -30492.411} C_VEL
LIN {X 0,Y 23.293,Z 447.684,A -85,B 0,C 180,E1 -30509.999,E2 -30509.999} C_VEL
LIN {X 0,Y 20.212,Z 451.701,A -85,B 0,C 180,E1 -30530.346,E2 -30530.346} C_VEL
LIN {X 0,Y 21.204,Z 456.492,A -85,B 0,C 180,E1 -30565.934,E2 -30565.934} C_VEL
LIN {X 0,Y 28.474,Z 459.902,A -85,B 0,C 180,E1 -30590.836,E2 -30590.836} C_VEL
LIN {X 0,Y 35.142,Z 461.486,A -85,B 0,C 180,E1 -30600.836,E2 -30600.836} C_VEL
LIN {X 0,Y 44.819,Z 462.662,A -85,B 0,C 180,E1 -30609.073,E2 -30609.073} C_VEL
LIN {X 0,Y 55.659,Z 462.903,A -85,B 0,C 180,E1 -30614.669,E2 -30614.669} C_VEL
LIN {X 0,Y 51.51,Z 463.094,A -85,B 0,C 180,E1 -30617.247,E2 -30617.247} C_VEL
LIN {X 0,Y 38.897,Z 462.631,A -85,B 0,C 180,E1 -30625.395,E2 -30625.395} C_VEL
LIN {X 0,Y 27.948,Z 460.762,A -85,B 0,C 180,E1 -30641.031,E2 -30641.031} C_VEL
LIN {X 0,Y 21.233,Z 457.424,A -85,B 0,C 180,E1 -30670.672,E2 -30670.672} C_VEL
LIN {X 0,Y 20.531,Z 455.057,A -85,B 0,C 180,E1 -30690.001,E2 -30690.001} C_VEL
LIN {X 0,Y 22.243,Z 450.4,A -85,B 0,C 180,E1 -30718.292,E2 -30718.292} C_VEL
LIN {X 0,Y 27.942,Z 444.436,A -85,B 0,C 180,E1 -30738.987,E2 -30738.987} C_VEL
LIN {X 0,Y 35.895,Z 436.973,A -85,B 0,C 180,E1 -30751.77,E2 -30751.77} C_VEL
LIN {X 0,Y 43.397,Z 429.348,A -85,B 0,C 180,E1 -30758.619,E2 -30758.619} C_VEL
LIN {X 0,Y 51.311,Z 420.065,A -85,B 0,C 180,E1 -30763.489,E2 -30763.489} C_VEL
LIN {X 0,Y 58.657,Z 409.73,A -85,B 0,C 180,E1 -30766.776,E2 -30766.776} C_VEL
LIN {X 0,Y 65.355,Z 398.424,A -85,B 0,C 180,E1 -30768.887,E2 -30768.887} C_VEL
LIN {X 0,Y 70.843,Z 386.686,A -85,B 0,C 180,E1 -30770.344,E2 -30770.344} C_VEL
LIN {X 0,Y 75.447,Z 373.307,A -85,B 0,C 180,E1 -30771.477,E2 -30771.477} C_VEL
LIN {X 0,Y 78.495,Z 360.69,A -85,B 0,C 180,E1 -30772.077,E2 -30772.077} C_VEL
LIN {X 0,Y 80.993,Z 342.84,A -85,B 0,C 180,E1 -30772.841,E2 -30772.841} C_VEL
LIN {X 0,Y 80.013,Z 338.831,A -85,B 0,C 180,E1 -30775.788,E2 -30775.788} C_VEL
LIN {X 0,Y 78.643,Z 333.765,A -85,B 0,C 180,E1 -30780.789,E2 -30780.789} C_VEL
LIN {X 0,Y 77.604,Z 329.91,A -85,B 0,C 180,E1 -30786.188,E2 -30786.188} C_VEL
LIN {X 0,Y 77.172,Z 328.242,A -85,B 0,C 180,E1 -30789.5,E2 -30789.5} C_VEL
LIN {X 0,Y 76.909,Z 326.73,A -85,B 0,C 180,E1 -30793.815,E2 -30793.815} C_VEL
LIN {X 0,Y 76.819,Z 326.893,A -85,B 0,C 180,E1 -30797.324,E2 -30797.324} C_VEL
LIN {X 0,Y 77.456,Z 330.318,A -85,B 0,C 180,E1 -30807.168,E2 -30807.168} C_VEL
LIN {X 0,Y 78.55,Z 333.855,A -85,B 0,C 180,E1 -30812.624,E2 -30812.624} C_VEL
LIN {X 0,Y 79.923,Z 338.38,A -85,B 0,C 180,E1 -30817.571,E2 -30817.571} C_VEL
LIN {X 0,Y 80.92,Z 341.832,A -85,B 0,C 180,E1 -30820.46,E2 -30820.46} C_VEL
LIN {X 0,Y 80.188,Z 347.914,A -85,B 0,C 180,E1 -30820.824,E2 -30820.824} C_VEL
LIN {X 0,Y 77.529,Z 363.462,A -85,B 0,C 180,E1 -30821.362,E2 -30821.362} C_VEL
LIN {X 0,Y 73.961,Z 376.537,A -85,B 0,C 180,E1 -30822.404,E2 -30822.404} C_VEL
LIN {X 0,Y 68.922,Z 389.566,A -85,B 0,C 180,E1 -30823.798,E2 -30823.798} C_VEL
LIN {X 0,Y 62.96,Z 401.322,A -85,B 0,C 180,E1 -30825.761,E2 -30825.761} C_VEL
LIN {X 0,Y 60.435,Z 405.577,A -85,B 0,C 180,E1 -30826.66,E2 -30826.66} C_VEL
LIN {X 0,Y 57.039,Z 410.367,A -85,B 0,C 180,E1 -30827.296,E2 -30827.296} C_VEL
LIN {X 0,Y 50.385,Z 417.71,A -85,B 0,C 180,E1 -30826.834,E2 -30826.834} C_VEL
LIN {X 0,Y 43.207,Z 424.584,A -85,B 0,C 180,E1 -30826.422,E2 -30826.422} C_VEL
LIN {X 0,Y 38.984,Z 428.645,A -85,B 0,C 180,E1 -30827.677,E2 -30827.677} C_VEL
LIN {X 0,Y 30.179,Z 436.808,A -85,B 0,C 180,E1 -30834.394,E2 -30834.394} C_VEL
LIN {X 0,Y 22.174,Z 443.363,A -85,B 0,C 180,E1 -30845.63,E2 -30845.63} C_VEL
LIN {X 0,Y 15.035,Z 449.269,A -85,B 0,C 180,E1 -30869.998,E2 -30869.998} C_VEL
LIN {X 0,Y 12.984,Z 454.322,A -85,B 0,C 180,E1 -30917.667,E2 -30917.667} C_VEL
LIN {X 0,Y 17.871,Z 457.584,A -85,B 0,C 180,E1 -30949.449,E2 -30949.449} C_VEL
LIN {X 0,Y 28.423,Z 460.76,A -85,B 0,C 180,E1 -30968.507,E2 -30968.507} C_VEL
LIN {X 0,Y 36.334,Z 462.12,A -85,B 0,C 180,E1 -30974.737,E2 -30974.737} C_VEL
LIN {X 0,Y 36.423,Z 462.144,A -85,B 0,C 180,E1 -30975.259,E2 -30975.259} C_VEL
LIN {X 0,Y 29.937,Z 461.285,A -85,B 0,C 180,E1 -30980.115,E2 -30980.115} C_VEL
LIN {X 0,Y 23.901,Z 460.09,A -85,B 0,C 180,E1 -30988.104,E2 -30988.104} C_VEL
LIN {X 0,Y 14.759,Z 456.485,A -85,B 0,C 180,E1 -31021.566,E2 -31021.566} C_VEL
LIN {X 0,Y 13.465,Z 454.029,A -85,B 0,C 180,E1 -31050.002,E2 -31050.002} C_VEL
LIN {X 0,Y 16.352,Z 449.18,A -85,B 0,C 180,E1 -31090.142,E2 -31090.142} C_VEL
LIN {X 0,Y 23.894,Z 442.997,A -85,B 0,C 180,E1 -31111.93,E2 -31111.93} C_VEL
LIN {X 0,Y 33.132,Z 435.229,A -85,B 0,C 180,E1 -31122.654,E2 -31122.654} C_VEL
LIN {X 0,Y 43.012,Z 425.496,A -85,B 0,C 180,E1 -31128.628,E2 -31128.628} C_VEL
LIN {X 0,Y 50.43,Z 416.706,A -85,B 0,C 180,E1 -31131.614,E2 -31131.614} C_VEL
LIN {X 0,Y 58.31,Z 405.375,A -85,B 0,C 180,E1 -31133.897,E2 -31133.897} C_VEL
LIN {X 0,Y 64.361,Z 394.627,A -85,B 0,C 180,E1 -31135.14,E2 -31135.14} C_VEL
LIN {X 0,Y 69.568,Z 382.912,A -85,B 0,C 180,E1 -31136.014,E2 -31136.014} C_VEL
LIN {X 0,Y 73.753,Z 370.144,A -85,B 0,C 180,E1 -31136.686,E2 -31136.686} C_VEL
LIN {X 0,Y 76.604,Z 356.807,A -85,B 0,C 180,E1 -31137.143,E2 -31137.143} C_VEL
LIN {X 0,Y 78.158,Z 345.511,A -85,B 0,C 180,E1 -31137.6,E2 -31137.6} C_VEL
LIN {X 0,Y 76.972,Z 339.871,A -85,B 0,C 180,E1 -31143.18,E2 -31143.18} C_VEL
LIN {X 0,Y 76.15,Z 335.722,A -85,B 0,C 180,E1 -31149.154,E2 -31149.154} C_VEL
LIN {X 0,Y 75.883,Z 333.81,A -85,B 0,C 180,E1 -31154.006,E2 -31154.006} C_VEL
LIN {X 0,Y 75.795,Z 333.975,A -85,B 0,C 180,E1 -31156.674,E2 -31156.674} C_VEL
LIN {X 0,Y 76.124,Z 336.87,A -85,B 0,C 180,E1 -31165.33,E2 -31165.33} C_VEL
LIN {X 0,Y 76.908,Z 340.063,A -85,B 0,C 180,E1 -31170.401,E2 -31170.401} C_VEL
LIN {X 0,Y 77.88,Z 344.087,A -85,B 0,C 180,E1 -31174.892,E2 -31174.892} C_VEL
LIN {X 0,Y 78.101,Z 345.462,A -85,B 0,C 180,E1 -31175.918,E2 -31175.918} C_VEL
LIN {X 0,Y 75.4,Z 361.895,A -85,B 0,C 180,E1 -31176.311,E2 -31176.311} C_VEL
LIN {X 0,Y 72.063,Z 374.671,A -85,B 0,C 180,E1 -31177.066,E2 -31177.066} C_VEL
LIN {X 0,Y 67.171,Z 387.513,A -85,B 0,C 180,E1 -31178.028,E2 -31178.028} C_VEL
LIN {X 0,Y 61.347,Z 399.212,A -85,B 0,C 180,E1 -31179.351,E2 -31179.351} C_VEL
LIN {X 0,Y 54.679,Z 409.887,A -85,B 0,C 180,E1 -31181.151,E2 -31181.151} C_VEL
LIN {X 0,Y 46.409,Z 420.573,A -85,B 0,C 180,E1 -31184.002,E2 -31184.002} C_VEL
LIN {X 0,Y 38.984,Z 428.645,A -85,B 0,C 180,E1 -31187.677,E2 -31187.677} C_VEL
LIN {X 0,Y 34.642,Z 432.524,A -85,B 0,C 180,E1 -31189.324,E2 -31189.324} C_VEL
LIN {X 0,Y 26.564,Z 438.256,A -85,B 0,C 180,E1 -31189.981,E2 -31189.981} C_VEL
LIN {X 0,Y 18.069,Z 443.457,A -85,B 0,C 180,E1 -31191.352,E2 -31191.352} C_VEL
LIN {X 0,Y 13.188,Z 446.432,A -85,B 0,C 180,E1 -31197.247,E2 -31197.247} C_VEL
LIN {X 0,Y 5.581,Z 452.687,A -85,B 0,C 180,E1 -31269.016,E2 -31269.016} C_VEL
LIN {X 0,Y 14.351,Z 457.365,A -85,B 0,C 180,E1 -31331.663,E2 -31331.663} C_VEL
LIN {X 0,Y 16.13,Z 457.946,A -85,B 0,C 180,E1 -31334.318,E2 -31334.318} C_VEL
LIN {X 0,Y 14.944,Z 457.629,A -85,B 0,C 180,E1 -31339.86,E2 -31339.86} C_VEL
LIN {X 0,Y 7.208,Z 454.304,A -85,B 0,C 180,E1 -31380.826,E2 -31380.826} C_VEL
LIN {X 0,Y 6.412,Z 452.963,A -85,B 0,C 180,E1 -31410.004,E2 -31410.004} C_VEL
LIN {X 0,Y 13.361,Z 446.881,A -85,B 0,C 180,E1 -31477.005,E2 -31477.005} C_VEL
LIN {X 0,Y 23.175,Z 440.183,A -85,B 0,C 180,E1 -31490.262,E2 -31490.262} C_VEL
LIN {X 0,Y 33.481,Z 431.847,A -85,B 0,C 180,E1 -31495.611,E2 -31495.611} C_VEL
LIN {X 0,Y 42.19,Z 423.24,A -85,B 0,C 180,E1 -31498.119,E2 -31498.119} C_VEL
LIN {X 0,Y 51.232,Z 412.24,A -85,B 0,C 180,E1 -31499.956,E2 -31499.956} C_VEL
LIN {X 0,Y 57.986,Z 402.172,A -85,B 0,C 180,E1 -31500.797,E2 -31500.797} C_VEL
LIN {X 0,Y 64.149,Z 390.648,A -85,B 0,C 180,E1 -31501.414,E2 -31501.414} C_VEL
LIN {X 0,Y 68.857,Z 379.238,A -85,B 0,C 180,E1 -31501.817,E2 -31501.817} C_VEL
LIN {X 0,Y 72.926,Z 365.634,A -85,B 0,C 180,E1 -31502.146,E2 -31502.146} C_VEL
LIN {X 0,Y 75.28,Z 352.98,A -85,B 0,C 180,E1 -31502.397,E2 -31502.397} C_VEL
LIN {X 0,Y 75.829,Z 348.861,A -85,B 0,C 180,E1 -31502.584,E2 -31502.584} C_VEL
LIN {X 0,Y 75.224,Z 344.918,A -85,B 0,C 180,E1 -31507.05,E2 -31507.05} C_VEL
LIN {X 0,Y 74.903,Z 342.037,A -85,B 0,C 180,E1 -31511.58,E2 -31511.58} C_VEL
LIN {X 0,Y 74.848,Z 341.35,A -85,B 0,C 180,E1 -31513.264,E2 -31513.264} C_VEL
LIN {X 0,Y 74.746,Z 341.297,A -85,B 0,C 180,E1 -31516.774,E2 -31516.774} C_VEL
LIN {X 0,Y 74.924,Z 343.799,A -85,B 0,C 180,E1 -31524.158,E2 -31524.158} C_VEL
LIN {X 0,Y 75.524,Z 347.126,A -85,B 0,C 180,E1 -31529.21,E2 -31529.21} C_VEL
LIN {X 0,Y 75.777,Z 348.515,A -85,B 0,C 180,E1 -31530.762,E2 -31530.762} C_VEL
LIN {X 0,Y 73.615,Z 361.458,A -85,B 0,C 180,E1 -31531.047,E2 -31531.047} C_VEL
LIN {X 0,Y 70.36,Z 373.929,A -85,B 0,C 180,E1 -31531.533,E2 -31531.533} C_VEL
LIN {X 0,Y 65.52,Z 386.723,A -85,B 0,C 180,E1 -31532.086,E2 -31532.086} C_VEL
LIN {X 0,Y 59.699,Z 398.367,A -85,B 0,C 180,E1 -31532.835,E2 -31532.835} C_VEL
LIN {X 0,Y 52.894,Z 409.186,A -85,B 0,C 180,E1 -31533.859,E2 -31533.859} C_VEL
LIN {X 0,Y 45.036,Z 419.299,A -85,B 0,C 180,E1 -31535.304,E2 -31535.304} C_VEL
LIN {X 0,Y 35.605,Z 429.163,A -85,B 0,C 180,E1 -31537.858,E2 -31537.858} C_VEL
LIN {X 0,Y 26.088,Z 437.374,A -85,B 0,C 180,E1 -31542.199,E2 -31542.199} C_VEL
LIN {X 0,Y 16.221,Z 444.482,A -85,B 0,C 180,E1 -31551.576,E2 -31551.576} C_VEL
LIN {X 0,Y 13.188,Z 446.432,A -85,B 0,C 180,E1 -31557.247,E2 -31557.247} C_VEL
LIN {X 0,Y 12.287,Z 446.676,A -85,B 0,C 180,E1 -31554.686,E2 -31554.686} C_VEL
LIN {X 0,Y 11.977,Z 446.156,A -85,B 0,C 180,E1 -31542.723,E2 -31542.723} C_VEL
LIN {X 0,Y 14.211,Z 444.317,A -85,B 0,C 180,E1 -31525.56,E2 -31525.56} C_VEL
LIN {X 0,Y 19.691,Z 440.661,A -85,B 0,C 180,E1 -31514.528,E2 -31514.528} C_VEL
LIN {X 0,Y 24.235,Z 437.48,A -85,B 0,C 180,E1 -31510.415,E2 -31510.415} C_VEL
LIN {X 0,Y 30.949,Z 432.211,A -85,B 0,C 180,E1 -31507.912,E2 -31507.912} C_VEL
LIN {X 0,Y 33.099,Z 430.305,A -85,B 0,C 180,E1 -31507.747,E2 -31507.747} C_VEL
LIN {X 0,Y 42.551,Z 420.8,A -85,B 0,C 180,E1 -31507.703,E2 -31507.703} C_VEL
LIN {X 0,Y 50.458,Z 411.016,A -85,B 0,C 180,E1 -31507.848,E2 -31507.848} C_VEL
LIN {X 0,Y 57.624,Z 400.057,A -85,B 0,C 180,E1 -31507.72,E2 -31507.72} C_VEL
LIN {X 0,Y 63.82,Z 388.022,A -85,B 0,C 180,E1 -31507.657,E2 -31507.657} C_VEL
LIN {X 0,Y 68.325,Z 376.568,A -85,B 0,C 180,E1 -31507.686,E2 -31507.686} C_VEL
LIN {X 0,Y 71.994,Z 363.518,A -85,B 0,C 180,E1 -31507.659,E2 -31507.659} C_VEL
LIN {X 0,Y 73.981,Z 352.36,A -85,B 0,C 180,E1 -31507.851,E2 -31507.851} C_VEL
LIN {X 0,Y 73.795,Z 348.752,A -85,B 0,C 180,E1 -31513.142,E2 -31513.142} C_VEL
LIN {X 0,Y 73.701,Z 348.614,A -85,B 0,C 180,E1 -31517.019,E2 -31517.019} C_VEL
LIN {X 0,Y 73.74,Z 350.516,A -85,B 0,C 180,E1 -31522.56,E2 -31522.56} C_VEL
LIN {X 0,Y 73.896,Z 352.636,A -85,B 0,C 180,E1 -31525.618,E2 -31525.618} C_VEL
LIN {X 0,Y 71.2,Z 366.14,A -85,B 0,C 180,E1 -31525.586,E2 -31525.586} C_VEL
LIN {X 0,Y 67.492,Z 378.383,A -85,B 0,C 180,E1 -31525.846,E2 -31525.846} C_VEL
LIN {X 0,Y 62.517,Z 390.349,A -85,B 0,C 180,E1 -31525.932,E2 -31525.932} C_VEL
LIN {X 0,Y 56.764,Z 401.096,A -85,B 0,C 180,E1 -31526.155,E2 -31526.155} C_VEL
LIN {X 0,Y 48.978,Z 412.591,A -85,B 0,C 180,E1 -31526.256,E2 -31526.256} C_VEL
LIN {X 0,Y 40.2,Z 423.041,A -85,B 0,C 180,E1 -31526.367,E2 -31526.367} C_VEL
LIN {X 0,Y 31.391,Z 431.579,A -85,B 0,C 180,E1 -31526.424,E2 -31526.424} C_VEL
LIN {X 0,Y 21.577,Z 439.384,A -85,B 0,C 180,E1 -31526.399,E2 -31526.399} C_VEL
LIN {X 0,Y 11.589,Z 445.873,A -85,B 0,C 180,E1 -31524.874,E2 -31524.874} C_VEL
LIN {X 0,Y 7.544,Z 448.154,A -85,B 0,C 180,E1 -31521.299,E2 -31521.299} C_VEL
LIN {X 0,Y 7.147,Z 448.415,A -85,B 0,C 180,E1 -31510.443,E2 -31510.443} C_VEL
LIN {X 0,Y 17.752,Z 442.196,A -85,B 0,C 180,E1 -31508.218,E2 -31508.218} C_VEL
LIN {X 0,Y 28.371,Z 434.384,A -85,B 0,C 180,E1 -31507.757,E2 -31507.757} C_VEL
LIN {X 0,Y 33.099,Z 430.305,A -85,B 0,C 180,E1 -31507.747,E2 -31507.747} C_VEL
LIN {X 0,Y 37.299,Z 426.227,A -85,B 0,C 180,E1 -31508.766,E2 -31508.766} C_VEL
LIN {X 0,Y 43.647,Z 418.996,A -85,B 0,C 180,E1 -31512.469,E2 -31512.469} C_VEL
LIN {X 0,Y 49.563,Z 411.321,A -85,B 0,C 180,E1 -31515.28,E2 -31515.28} C_VEL
LIN {X 0,Y 52.915,Z 406.437,A -85,B 0,C 180,E1 -31515.477,E2 -31515.477} C_VEL
LIN {X 0,Y 58.994,Z 396.306,A -85,B 0,C 180,E1 -31514.552,E2 -31514.552} C_VEL
LIN {X 0,Y 64.787,Z 383.982,A -85,B 0,C 180,E1 -31513.829,E2 -31513.829} C_VEL
LIN {X 0,Y 69.482,Z 370.457,A -85,B 0,C 180,E1 -31513.454,E2 -31513.454} C_VEL
LIN {X 0,Y 72.387,Z 357.871,A -85,B 0,C 180,E1 -31513.238,E2 -31513.238} C_VEL
LIN {X 0,Y 72.629,Z 356.342,A -85,B 0,C 180,E1 -31513.41,E2 -31513.41} C_VEL
LIN {X 0,Y 72.683,Z 355.591,A -85,B 0,C 180,E1 -31514.779,E2 -31514.779} C_VEL
LIN {X 0,Y 72.619,Z 355.804,A -85,B 0,C 180,E1 -31516.844,E2 -31516.844} C_VEL
LIN {X 0,Y 72.556,Z 356.677,A -85,B 0,C 180,E1 -31519.885,E2 -31519.885} C_VEL
LIN {X 0,Y 69.526,Z 370.149,A -85,B 0,C 180,E1 -31519.909,E2 -31519.909} C_VEL
LIN {X 0,Y 65.354,Z 382.441,A -85,B 0,C 180,E1 -31519.745,E2 -31519.745} C_VEL
LIN {X 0,Y 59.557,Z 395.136,A -85,B 0,C 180,E1 -31519.261,E2 -31519.261} C_VEL
LIN {X 0,Y 52.805,Z 406.563,A -85,B 0,C 180,E1 -31518.543,E2 -31518.543} C_VEL
LIN {X 0,Y 44.112,Z 418.202,A -85,B 0,C 180,E1 -31517.075,E2 -31517.075} C_VEL
LIN {X 0,Y 52.143,Z 407.565,A -85,B 0,C 180,E1 -31515.592,E2 -31515.592} C_VEL
LIN {X 0,Y 52.915,Z 406.437,A -85,B 0,C 180,E1 -31515.477,E2 -31515.477} C_VEL
LIN {X 0,Y 56.539,Z 407.54,A -85,B 0,C 180,E1 -31514.884,E2 -31514.884} C_VEL
LIN {X 0,Y 56.539,Z 600,A -85,B 0,C 180,E1 -31514.884,E2 -31514.884} C_VEL
LIN {X 0,Y 56.539,Z 600,A -85,B 0,C 180,E1 -31514.884,E2 -31514.884}

QRS_NEXT_CUT()

QRS_NEXT()
QRS_HOME()

END
